KUKA KRL program: EPS_2_251349_MH90A_A_20250929014703.src

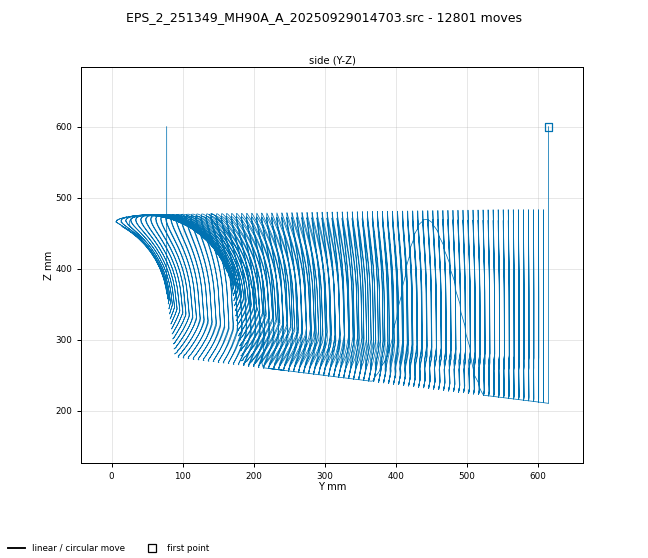
[picture p0: tool path of EPS_2_251349_MH90A_A_20250929014703.src, 12801 of 12803 moves have a stored position in this frame; points joined in program order, loops and branches not executed]
&ACCESS RVP
&REL 4
&COMMENT QRS 19112012
&PARAM EDITMASK = *
DEF PART()
EXT BAS (BAS_COMMAND :IN,REAL :IN )
INT I
BAS (#INITMOV,0 )

;KUKA QRS Post kuka4.cps  Date:22-06-2017 !

File_ID=2864

QRS_PRE_INIT()

;Init var - Until changes are made in qrs_pre_init
Outlet_Square_prg=0
Inlet_1_Square_prg=0
Inlet_2_Square_prg=0
Inlet_3_Square_prg=0
Inlet_4_Square_prg=0
Inlet_5_Square_prg=0

Outlet_1={X 0.000, Y 540.910, Z 382.500, B 0.000, E1 0.000 }
Inlet_1={X 0.000, Y 541.980, Z 367.500, B 0.000, E1 159.000 }
Outlet_1_type=201
Inlet_1_type=201
;QRS#1=Sidecore dimensions
;QRS#2=200-8" PVC SDR 35
;QRS#3=200-8" PVC SDR 35
;QRS#4=
;QRS#5=
;QRS#6=
;QRS#7=
;QRS#8=
;QRS#9=12-08 PSX
;QRS#10=12-08 PSX
;QRS#11=
;QRS#12=
;QRS#13=
;QRS#14=
;QRS#15=
;QRS#16=1220x127x762 2,5'
;QRS#17=EPS Height
;QRS#18=483
;QRS#19=*
;QRS#20= UPDATED VERSION 22-06-2017
;QRS#21=*
Outlet_Square=0100
Inlet_1_Square=0100
Inlet_2_Square=0
Inlet_3_Square=0
Inlet_4_Square=0
Inlet_5_Square=0
Mill_Square=1
Outlet_Square_Prg=204
Inlet_1_Square_prg=204

QRS_INIT()

$ADVANCE=5

; T1
PTP {E1 173.658,E2 173.658}
PTP {X 0,Y 615.42,A -85,B 0,C 180,E1 173.658,E2 173.658,E3 0,E4 0,E5 0,E6 0}
QRS_SPEED_INIT()
LIN {X 0,Y 615.42,Z 600,A -85,B 0,C 180,E1 173.658,E2 173.658,E3 0,E4 0,E5 0,E6 0} C_VEL
LIN {X 0,Y 615.42,Z 220.377,A -85,B 0,C 180,E1 173.658,E2 173.658} C_VEL
LIN {X 0,Y 615.42,Z 212.199,A -85,B 0,C 180,E1 173.658,E2 173.658} C_VEL
LIN {X 0,Y 615.409,Z 210.199,A -85,B 0,C 180,E1 173.472,E2 173.472} C_VEL
LIN {X 0,Y 615.414,Z 210.198,A -85,B 0,C 180,E1 171.465,E2 171.465} C_VEL
LIN {X 0,Y 615.421,Z 210.198,A -85,B 0,C 180,E1 169.475,E2 169.475} C_VEL
LIN {X 0,Y 615.428,Z 210.197,A -85,B 0,C 180,E1 167.472,E2 167.472} C_VEL
LIN {X 0,Y 615.434,Z 210.196,A -85,B 0,C 180,E1 165.453,E2 165.453} C_VEL
LIN {X 0,Y 615.439,Z 210.195,A -85,B 0,C 180,E1 163.415,E2 163.415} C_VEL
LIN {X 0,Y 615.442,Z 210.195,A -85,B 0,C 180,E1 161.356,E2 161.356} C_VEL
LIN {X 0,Y 615.442,Z 210.194,A -85,B 0,C 180,E1 159.271,E2 159.271} C_VEL
LIN {X 0,Y 615.441,Z 210.193,A -85,B 0,C 180,E1 157.157,E2 157.157} C_VEL
LIN {X 0,Y 615.437,Z 210.193,A -85,B 0,C 180,E1 155.01,E2 155.01} C_VEL
LIN {X 0,Y 615.432,Z 210.193,A -85,B 0,C 180,E1 152.824,E2 152.824} C_VEL
LIN {X 0,Y 615.429,Z 210.194,A -85,B 0,C 180,E1 150.595,E2 150.595} C_VEL
LIN {X 0,Y 615.43,Z 210.195,A -85,B 0,C 180,E1 148.316,E2 148.316} C_VEL
LIN {X 0,Y 615.446,Z 210.197,A -85,B 0,C 180,E1 145.98,E2 145.98} C_VEL
LIN {X 0,Y 615.487,Z 210.189,A -85,B 0,C 180,E1 143.061,E2 143.061} C_VEL
LIN {X 0,Y 615.489,Z 210.187,A -85,B 0,C 180,E1 140.935,E2 140.935} C_VEL
LIN {X 0,Y 615.457,Z 210.188,A -85,B 0,C 180,E1 138.529,E2 138.529} C_VEL
LIN {X 0,Y 615.441,Z 210.192,A -85,B 0,C 180,E1 136.005,E2 136.005} C_VEL
LIN {X 0,Y 615.49,Z 210.199,A -85,B 0,C 180,E1 133.243,E2 133.243} C_VEL
LIN {X 0,Y 615.493,Z 210.363,A -85,B 0,C 180,E1 131.038,E2 131.038} C_VEL
LIN {X 0,Y 615.491,Z 226.448,A -85,B 0,C 180,E1 128.483,E2 128.483} C_VEL
LIN {X 0,Y 615.431,Z 244.942,A -85,B 0,C 180,E1 125.618,E2 125.618} C_VEL
LIN {X 0,Y 615.451,Z 256.457,A -85,B 0,C 180,E1 123.87,E2 123.87} C_VEL
LIN {X 0,Y 615.447,Z 258.462,A -85,B 0,C 180,E1 123.794,E2 123.794} C_VEL
LIN {X 0,Y 615.497,Z 363.346,A -85,B 0,C 180,E1 122.552,E2 122.552} C_VEL
LIN {X 0,Y 615.5,Z 376.884,A -85,B 0,C 180,E1 122.258,E2 122.258} C_VEL
LIN {X 0,Y 615.498,Z 389.472,A -85,B 0,C 180,E1 121.847,E2 121.847} C_VEL
LIN {X 0,Y 615.478,Z 401.528,A -85,B 0,C 180,E1 121.313,E2 121.313} C_VEL
LIN {X 0,Y 615.477,Z 413.275,A -85,B 0,C 180,E1 120.633,E2 120.633} C_VEL
LIN {X 0,Y 615.497,Z 423.488,A -85,B 0,C 180,E1 119.894,E2 119.894} C_VEL
LIN {X 0,Y 615.497,Z 431.12,A -85,B 0,C 180,E1 119.217,E2 119.217} C_VEL
LIN {X 0,Y 615.497,Z 439.703,A -85,B 0,C 180,E1 118.324,E2 118.324} C_VEL
LIN {X 0,Y 615.488,Z 447.119,A -85,B 0,C 180,E1 117.36,E2 117.36} C_VEL
LIN {X 0,Y 615.496,Z 452.856,A -85,B 0,C 180,E1 116.442,E2 116.442} C_VEL
LIN {X 0,Y 615.495,Z 458.535,A -85,B 0,C 180,E1 115.285,E2 115.285} C_VEL
LIN {X 0,Y 615.496,Z 462.263,A -85,B 0,C 180,E1 114.27,E2 114.27} C_VEL
LIN {X 0,Y 615.494,Z 464.278,A -85,B 0,C 180,E1 113.555,E2 113.555} C_VEL
LIN {X 0,Y 615.492,Z 466.468,A -85,B 0,C 180,E1 112.359,E2 112.359} C_VEL
LIN {X 0,Y 615.497,Z 467.282,A -85,B 0,C 180,E1 111.43,E2 111.43} C_VEL
LIN {X 0,Y 615.494,Z 467.304,A -85,B 0,C 180,E1 110.572,E2 110.572} C_VEL
LIN {X 0,Y 615.496,Z 466.182,A -85,B 0,C 180,E1 109.336,E2 109.336} C_VEL
LIN {X 0,Y 615.496,Z 464.861,A -85,B 0,C 180,E1 108.622,E2 108.622} C_VEL
LIN {X 0,Y 615.499,Z 462.172,A -85,B 0,C 180,E1 107.612,E2 107.612} C_VEL
LIN {X 0,Y 615.495,Z 457.783,A -85,B 0,C 180,E1 106.45,E2 106.45} C_VEL
LIN {X 0,Y 615.497,Z 453.383,A -85,B 0,C 180,E1 105.564,E2 105.564} C_VEL
LIN {X 0,Y 615.489,Z 447.102,A -85,B 0,C 180,E1 104.548,E2 104.548} C_VEL
LIN {X 0,Y 615.5,Z 439.266,A -85,B 0,C 180,E1 103.536,E2 103.536} C_VEL
LIN {X 0,Y 615.496,Z 429.44,A -85,B 0,C 180,E1 102.529,E2 102.529} C_VEL
LIN {X 0,Y 615.498,Z 420.424,A -85,B 0,C 180,E1 101.776,E2 101.776} C_VEL
LIN {X 0,Y 615.475,Z 409.654,A -85,B 0,C 180,E1 101.049,E2 101.049} C_VEL
LIN {X 0,Y 615.492,Z 398.322,A -85,B 0,C 180,E1 100.443,E2 100.443} C_VEL
LIN {X 0,Y 615.498,Z 386.276,A -85,B 0,C 180,E1 99.944,E2 99.944} C_VEL
LIN {X 0,Y 615.498,Z 373.8,A -85,B 0,C 180,E1 99.57,E2 99.57} C_VEL
LIN {X 0,Y 615.497,Z 360.801,A -85,B 0,C 180,E1 99.322,E2 99.322} C_VEL
LIN {X 0,Y 615.431,Z 257.063,A -85,B 0,C 180,E1 98.082,E2 98.082} C_VEL
LIN {X 0,Y 615.443,Z 255.243,A -85,B 0,C 180,E1 97.875,E2 97.875} C_VEL
LIN {X 0,Y 615.472,Z 235.998,A -85,B 0,C 180,E1 94.912,E2 94.912} C_VEL
LIN {X 0,Y 615.489,Z 218.149,A -85,B 0,C 180,E1 92.126,E2 92.126} C_VEL
LIN {X 0,Y 615.493,Z 210.327,A -85,B 0,C 180,E1 90.858,E2 90.858} C_VEL
LIN {X 0,Y 615.425,Z 210.197,A -85,B 0,C 180,E1 88.036,E2 88.036} C_VEL
LIN {X 0,Y 615.43,Z 210.198,A -85,B 0,C 180,E1 86.07,E2 86.07} C_VEL
LIN {X 0,Y 615.436,Z 210.198,A -85,B 0,C 180,E1 84.1,E2 84.1} C_VEL
LIN {X 0,Y 615.444,Z 210.199,A -85,B 0,C 180,E1 82.123,E2 82.123} C_VEL
LIN {X 0,Y 615.449,Z 210.2,A -85,B 0,C 180,E1 80.136,E2 80.136} C_VEL
LIN {X 0,Y 615.413,Z 210.197,A -85,B 0,C 180,E1 77.467,E2 77.467} C_VEL
LIN {X 0,Y 615.414,Z 210.198,A -85,B 0,C 180,E1 75.448,E2 75.448} C_VEL
LIN {X 0,Y 615.411,Z 210.198,A -85,B 0,C 180,E1 73.41,E2 73.41} C_VEL
LIN {X 0,Y 615.412,Z 210.198,A -85,B 0,C 180,E1 71.351,E2 71.351} C_VEL
LIN {X 0,Y 615.411,Z 210.198,A -85,B 0,C 180,E1 69.266,E2 69.266} C_VEL
LIN {X 0,Y 615.409,Z 210.199,A -85,B 0,C 180,E1 67.152,E2 67.152} C_VEL
LIN {X 0,Y 615.407,Z 210.199,A -85,B 0,C 180,E1 65.004,E2 65.004} C_VEL
LIN {X 0,Y 615.404,Z 210.199,A -85,B 0,C 180,E1 62.818,E2 62.818} C_VEL
LIN {X 0,Y 615.442,Z 210.199,A -85,B 0,C 180,E1 60.204,E2 60.204} C_VEL
LIN {X 0,Y 615.467,Z 210.2,A -85,B 0,C 180,E1 57.54,E2 57.54} C_VEL
LIN {X 0,Y 615.43,Z 210.2,A -85,B 0,C 180,E1 55.18,E2 55.18} C_VEL
LIN {X 0,Y 615.405,Z 210.2,A -85,B 0,C 180,E1 52.751,E2 52.751} C_VEL
LIN {X 0,Y 615.408,Z 210.2,A -85,B 0,C 180,E1 50.243,E2 50.243} C_VEL
LIN {X 0,Y 615.426,Z 210.2,A -85,B 0,C 180,E1 47.92,E2 47.92} C_VEL
LIN {X 0,Y 615.448,Z 210.198,A -85,B 0,C 180,E1 44.927,E2 44.927} C_VEL
LIN {X 0,Y 615.473,Z 210.198,A -85,B 0,C 180,E1 43.045,E2 43.045} C_VEL
LIN {X 0,Y 615.432,Z 210.197,A -85,B 0,C 180,E1 40.606,E2 40.606} C_VEL
LIN {X 0,Y 615.48,Z 210.196,A -85,B 0,C 180,E1 38.9,E2 38.9} C_VEL
LIN {X 0,Y 615.432,Z 210.197,A -85,B 0,C 180,E1 36.424,E2 36.424} C_VEL
LIN {X 0,Y 615.414,Z 210.197,A -85,B 0,C 180,E1 34.022,E2 34.022} C_VEL
LIN {X 0,Y 615.415,Z 210.198,A -85,B 0,C 180,E1 31.685,E2 31.685} C_VEL
LIN {X 0,Y 615.423,Z 210.198,A -85,B 0,C 180,E1 29.405,E2 29.405} C_VEL
LIN {X 0,Y 615.453,Z 210.199,A -85,B 0,C 180,E1 27.037,E2 27.037} C_VEL
LIN {X 0,Y 615.44,Z 210.194,A -85,B 0,C 180,E1 23.997,E2 23.997} C_VEL
LIN {X 0,Y 615.464,Z 210.193,A -85,B 0,C 180,E1 22.134,E2 22.134} C_VEL
LIN {X 0,Y 615.462,Z 210.193,A -85,B 0,C 180,E1 20.03,E2 20.03} C_VEL
LIN {X 0,Y 615.459,Z 210.193,A -85,B 0,C 180,E1 17.954,E2 17.954} C_VEL
LIN {X 0,Y 615.467,Z 210.192,A -85,B 0,C 180,E1 15.902,E2 15.902} C_VEL
LIN {X 0,Y 615.425,Z 210.195,A -85,B 0,C 180,E1 13.199,E2 13.199} C_VEL
LIN {X 0,Y 615.426,Z 210.197,A -85,B 0,C 180,E1 10.856,E2 10.856} C_VEL
LIN {X 0,Y 615.446,Z 210.197,A -85,B 0,C 180,E1 8.534,E2 8.534} C_VEL
LIN {X 0,Y 615.497,Z 210.195,A -85,B 0,C 180,E1 5.896,E2 5.896} C_VEL
LIN {X 0,Y 615.453,Z 210.19,A -85,B 0,C 180,E1 3.27,E2 3.27} C_VEL
LIN {X 0,Y 615.466,Z 210.189,A -85,B 0,C 180,E1 1.306,E2 1.306} C_VEL
LIN {X 0,Y 615.432,Z 210.193,A -85,B 0,C 180,E1 -1.311,E2 -1.311} C_VEL
LIN {X 0,Y 615.436,Z 210.192,A -85,B 0,C 180,E1 -3.276,E2 -3.276} C_VEL
LIN {X 0,Y 615.441,Z 210.191,A -85,B 0,C 180,E1 -5.244,E2 -5.244} C_VEL
LIN {X 0,Y 615.449,Z 210.19,A -85,B 0,C 180,E1 -7.218,E2 -7.218} C_VEL
LIN {X 0,Y 615.457,Z 210.189,A -85,B 0,C 180,E1 -9.201,E2 -9.201} C_VEL
LIN {X 0,Y 615.466,Z 210.188,A -85,B 0,C 180,E1 -11.196,E2 -11.196} C_VEL
LIN {X 0,Y 615.472,Z 210.187,A -85,B 0,C 180,E1 -13.204,E2 -13.204} C_VEL
LIN {X 0,Y 615.439,Z 210.192,A -85,B 0,C 180,E1 -15.908,E2 -15.908} C_VEL
LIN {X 0,Y 615.475,Z 210.199,A -85,B 0,C 180,E1 -18.6,E2 -18.6} C_VEL
LIN {X 0,Y 615.485,Z 210.185,A -85,B 0,C 180,E1 -21.434,E2 -21.434} C_VEL
LIN {X 0,Y 615.446,Z 210.19,A -85,B 0,C 180,E1 -23.998,E2 -23.998} C_VEL
LIN {X 0,Y 615.447,Z 210.194,A -85,B 0,C 180,E1 -26.448,E2 -26.448} C_VEL
LIN {X 0,Y 615.493,Z 210.19,A -85,B 0,C 180,E1 -29.408,E2 -29.408} C_VEL
LIN {X 0,Y 615.489,Z 210.186,A -85,B 0,C 180,E1 -31.687,E2 -31.687} C_VEL
LIN {X 0,Y 615.474,Z 210.185,A -85,B 0,C 180,E1 -34.024,E2 -34.024} C_VEL
LIN {X 0,Y 615.453,Z 210.188,A -85,B 0,C 180,E1 -36.429,E2 -36.429} C_VEL
LIN {X 0,Y 615.461,Z 210.195,A -85,B 0,C 180,E1 -39.058,E2 -39.058} C_VEL
LIN {X 0,Y 615.491,Z 210.201,A -85,B 0,C 180,E1 -41.475,E2 -41.475} C_VEL
LIN {X 0,Y 615.496,Z 210.183,A -85,B 0,C 180,E1 -44.15,E2 -44.15} C_VEL
LIN {X 0,Y 615.454,Z 210.19,A -85,B 0,C 180,E1 -46.957,E2 -46.957} C_VEL
LIN {X 0,Y 615.464,Z 210.195,A -85,B 0,C 180,E1 -49.391,E2 -49.391} C_VEL
LIN {X 0,Y 615.49,Z 210.197,A -85,B 0,C 180,E1 -51.989,E2 -51.989} C_VEL
LIN {X 0,Y 615.489,Z 210.187,A -85,B 0,C 180,E1 -54.383,E2 -54.383} C_VEL
LIN {X 0,Y 615.486,Z 210.182,A -85,B 0,C 180,E1 -56.763,E2 -56.763} C_VEL
LIN {X 0,Y 615.472,Z 210.184,A -85,B 0,C 180,E1 -59.079,E2 -59.079} C_VEL
LIN {X 0,Y 615.46,Z 210.19,A -85,B 0,C 180,E1 -61.556,E2 -61.556} C_VEL
LIN {X 0,Y 615.498,Z 210.199,A -85,B 0,C 180,E1 -64.284,E2 -64.284} C_VEL
LIN {X 0,Y 615.484,Z 210.182,A -85,B 0,C 180,E1 -67.154,E2 -67.154} C_VEL
LIN {X 0,Y 615.492,Z 210.435,A -85,B 0,C 180,E1 -68.48,E2 -68.48} C_VEL
LIN {X 0,Y 615.494,Z 228.954,A -85,B 0,C 180,E1 -71.181,E2 -71.181} C_VEL
LIN {X 0,Y 615.488,Z 249.417,A -85,B 0,C 180,E1 -74.094,E2 -74.094} C_VEL
LIN {X 0,Y 615.473,Z 268.657,A -85,B 0,C 180,E1 -76.798,E2 -76.798} C_VEL
LIN {X 0,Y 615.487,Z 271.231,A -85,B 0,C 180,E1 -77.113,E2 -77.113} C_VEL
LIN {X 0,Y 615.49,Z 278.177,A -85,B 0,C 180,E1 -77.218,E2 -77.218} C_VEL
LIN {X 0,Y 615.498,Z 378.775,A -85,B 0,C 180,E1 -78.41,E2 -78.41} C_VEL
LIN {X 0,Y 615.498,Z 391.308,A -85,B 0,C 180,E1 -78.681,E2 -78.681} C_VEL
LIN {X 0,Y 615.496,Z 404.514,A -85,B 0,C 180,E1 -79.109,E2 -79.109} C_VEL
LIN {X 0,Y 615.491,Z 416.458,A -85,B 0,C 180,E1 -79.639,E2 -79.639} C_VEL
LIN {X 0,Y 615.48,Z 427.982,A -85,B 0,C 180,E1 -80.303,E2 -80.303} C_VEL
LIN {X 0,Y 615.499,Z 438.329,A -85,B 0,C 180,E1 -81.049,E2 -81.049} C_VEL
LIN {X 0,Y 615.498,Z 446.682,A -85,B 0,C 180,E1 -81.793,E2 -81.793} C_VEL
LIN {X 0,Y 615.498,Z 454.598,A -85,B 0,C 180,E1 -82.619,E2 -82.619} C_VEL
LIN {X 0,Y 615.49,Z 462.198,A -85,B 0,C 180,E1 -83.607,E2 -83.607} C_VEL
LIN {X 0,Y 615.498,Z 469.199,A -85,B 0,C 180,E1 -84.758,E2 -84.758} C_VEL
LIN {X 0,Y 615.493,Z 473.847,A -85,B 0,C 180,E1 -85.743,E2 -85.743} C_VEL
LIN {X 0,Y 615.494,Z 477.396,A -85,B 0,C 180,E1 -86.726,E2 -86.726} C_VEL
LIN {X 0,Y 615.497,Z 479.23,A -85,B 0,C 180,E1 -87.381,E2 -87.381} C_VEL
LIN {X 0,Y 615.497,Z 480.606,A -85,B 0,C 180,E1 -88.036,E2 -88.036} C_VEL
LIN {X 0,Y 615.496,Z 482.173,A -85,B 0,C 180,E1 -89.345,E2 -89.345} C_VEL
LIN {X 0,Y 615.494,Z 482.389,A -85,B 0,C 180,E1 -89.999,E2 -89.999} C_VEL
LIN {X 0,Y 615.495,Z 481.581,A -85,B 0,C 180,E1 -91.308,E2 -91.308} C_VEL
LIN {X 0,Y 615.497,Z 480.61,A -85,B 0,C 180,E1 -91.962,E2 -91.962} C_VEL
LIN {X 0,Y 615.497,Z 479.236,A -85,B 0,C 180,E1 -92.617,E2 -92.617} C_VEL
LIN {X 0,Y 615.496,Z 476.353,A -85,B 0,C 180,E1 -93.6,E2 -93.6} C_VEL
LIN {X 0,Y 615.498,Z 472.446,A -85,B 0,C 180,E1 -94.583,E2 -94.583} C_VEL
LIN {X 0,Y 615.499,Z 467.411,A -85,B 0,C 180,E1 -95.569,E2 -95.569} C_VEL
LIN {X 0,Y 615.489,Z 460.919,A -85,B 0,C 180,E1 -96.577,E2 -96.577} C_VEL
LIN {X 0,Y 615.497,Z 453.143,A -85,B 0,C 180,E1 -97.544,E2 -97.544} C_VEL
LIN {X 0,Y 615.498,Z 443.27,A -85,B 0,C 180,E1 -98.535,E2 -98.535} C_VEL
LIN {X 0,Y 615.495,Z 432.881,A -85,B 0,C 180,E1 -99.363,E2 -99.363} C_VEL
LIN {X 0,Y 615.475,Z 422.596,A -85,B 0,C 180,E1 -100.027,E2 -100.027} C_VEL
LIN {X 0,Y 615.497,Z 411.116,A -85,B 0,C 180,E1 -100.617,E2 -100.617} C_VEL
LIN {X 0,Y 615.499,Z 399.293,A -85,B 0,C 180,E1 -101.079,E2 -101.079} C_VEL
LIN {X 0,Y 615.498,Z 386.288,A -85,B 0,C 180,E1 -101.442,E2 -101.442} C_VEL
LIN {X 0,Y 615.5,Z 373.028,A -85,B 0,C 180,E1 -101.671,E2 -101.671} C_VEL
LIN {X 0,Y 615.488,Z 271.775,A -85,B 0,C 180,E1 -102.864,E2 -102.864} C_VEL
LIN {X 0,Y 615.485,Z 270.528,A -85,B 0,C 180,E1 -102.948,E2 -102.948} C_VEL
LIN {X 0,Y 615.481,Z 250.635,A -85,B 0,C 180,E1 -105.734,E2 -105.734} C_VEL
LIN {X 0,Y 615.491,Z 231.587,A -85,B 0,C 180,E1 -108.442,E2 -108.442} C_VEL
LIN {X 0,Y 615.493,Z 212.1,A -85,B 0,C 180,E1 -111.255,E2 -111.255} C_VEL
LIN {X 0,Y 615.49,Z 210.316,A -85,B 0,C 180,E1 -111.562,E2 -111.562} C_VEL
LIN {X 0,Y 615.461,Z 210.19,A -85,B 0,C 180,E1 -114.272,E2 -114.272} C_VEL
LIN {X 0,Y 615.497,Z 210.18,A -85,B 0,C 180,E1 -117.046,E2 -117.046} C_VEL
LIN {X 0,Y 615.497,Z 210.199,A -85,B 0,C 180,E1 -119.795,E2 -119.795} C_VEL
LIN {X 0,Y 615.457,Z 210.192,A -85,B 0,C 180,E1 -122.458,E2 -122.458} C_VEL
LIN {X 0,Y 615.455,Z 210.188,A -85,B 0,C 180,E1 -124.816,E2 -124.816} C_VEL
LIN {X 0,Y 615.476,Z 210.184,A -85,B 0,C 180,E1 -127.241,E2 -127.241} C_VEL
LIN {X 0,Y 615.498,Z 210.199,A -85,B 0,C 180,E1 -130.089,E2 -130.089} C_VEL
LIN {X 0,Y 615.48,Z 210.198,A -85,B 0,C 180,E1 -132.352,E2 -132.352} C_VEL
LIN {X 0,Y 615.443,Z 210.192,A -85,B 0,C 180,E1 -135.071,E2 -135.071} C_VEL
LIN {X 0,Y 615.498,Z 210.185,A -85,B 0,C 180,E1 -137.917,E2 -137.917} C_VEL
LIN {X 0,Y 615.495,Z 210.195,A -85,B 0,C 180,E1 -140.249,E2 -140.249} C_VEL
LIN {X 0,Y 615.443,Z 210.195,A -85,B 0,C 180,E1 -143.066,E2 -143.066} C_VEL
LIN {X 0,Y 615.437,Z 210.193,A -85,B 0,C 180,E1 -145.304,E2 -145.304} C_VEL
LIN {X 0,Y 615.44,Z 210.191,A -85,B 0,C 180,E1 -147.673,E2 -147.673} C_VEL
LIN {X 0,Y 615.491,Z 210.198,A -85,B 0,C 180,E1 -150.592,E2 -150.592} C_VEL
LIN {X 0,Y 615.473,Z 210.199,A -85,B 0,C 180,E1 -152.954,E2 -152.954} C_VEL
LIN {X 0,Y 615.473,Z 210.199,A -85,B 0,C 180,E1 -155.006,E2 -155.006} C_VEL
LIN {X 0,Y 615.427,Z 210.196,A -85,B 0,C 180,E1 -157.664,E2 -157.664} C_VEL
LIN {X 0,Y 615.423,Z 210.195,A -85,B 0,C 180,E1 -159.963,E2 -159.963} C_VEL
LIN {X 0,Y 615.48,Z 210.193,A -85,B 0,C 180,E1 -162.727,E2 -162.727} C_VEL
LIN {X 0,Y 615.452,Z 210.199,A -85,B 0,C 180,E1 -165.448,E2 -165.448} C_VEL
LIN {X 0,Y 615.455,Z 210.199,A -85,B 0,C 180,E1 -167.467,E2 -167.467} C_VEL
LIN {X 0,Y 615.462,Z 210.199,A -85,B 0,C 180,E1 -169.47,E2 -169.47} C_VEL
LIN {X 0,Y 615.413,Z 210.198,A -85,B 0,C 180,E1 -172.121,E2 -172.121} C_VEL
LIN {X 0,Y 615.413,Z 210.199,A -85,B 0,C 180,E1 -174.098,E2 -174.098} C_VEL
LIN {X 0,Y 615.417,Z 210.199,A -85,B 0,C 180,E1 -176.069,E2 -176.069} C_VEL
LIN {X 0,Y 615.419,Z 210.2,A -85,B 0,C 180,E1 -178.034,E2 -178.034} C_VEL
LIN {X 0,Y 615.43,Z 210.2,A -85,B 0,C 180,E1 -179.997,E2 -179.997} C_VEL
LIN {X 0,Y 615.44,Z 210.2,A -85,B 0,C 180,E1 -181.961,E2 -181.961} C_VEL
LIN {X 0,Y 615.404,Z 210.2,A -85,B 0,C 180,E1 -184.582,E2 -184.582} C_VEL
LIN {X 0,Y 615.409,Z 210.199,A -85,B 0,C 180,E1 -186.528,E2 -186.528} C_VEL
LIN {X 0,Y 614.74,Z 210.347,A -85,B 0,C 180,E1 -187.074,E2 -187.074} C_VEL
LIN {X 0,Y 611.905,Z 210.764,A -85,B 0,C 180,E1 -187.961,E2 -187.961} C_VEL
LIN {X 0,Y 609.519,Z 211.07,A -85,B 0,C 180,E1 -188.673,E2 -188.673} C_VEL
LIN {X 0,Y 608.5,Z 211.185,A -85,B 0,C 180,E1 -189.223,E2 -189.223} C_VEL
LIN {X 0,Y 608.42,Z 211.194,A -85,B 0,C 180,E1 -189.409,E2 -189.409} C_VEL
LIN {X 0,Y 608.446,Z 211.196,A -85,B 0,C 180,E1 -191.997,E2 -191.997} C_VEL
LIN {X 0,Y 608.393,Z 211.194,A -85,B 0,C 180,E1 -194.719,E2 -194.719} C_VEL
LIN {X 0,Y 608.401,Z 211.193,A -85,B 0,C 180,E1 -196.782,E2 -196.782} C_VEL
LIN {X 0,Y 608.415,Z 211.191,A -85,B 0,C 180,E1 -198.867,E2 -198.867} C_VEL
LIN {X 0,Y 608.411,Z 211.192,A -85,B 0,C 180,E1 -200.98,E2 -200.98} C_VEL
LIN {X 0,Y 608.403,Z 211.193,A -85,B 0,C 180,E1 -203.122,E2 -203.122} C_VEL
LIN {X 0,Y 608.396,Z 211.193,A -85,B 0,C 180,E1 -205.3,E2 -205.3} C_VEL
LIN {X 0,Y 608.407,Z 211.193,A -85,B 0,C 180,E1 -207.516,E2 -207.516} C_VEL
LIN {X 0,Y 608.428,Z 211.194,A -85,B 0,C 180,E1 -209.968,E2 -209.968} C_VEL
LIN {X 0,Y 608.437,Z 211.192,A -85,B 0,C 180,E1 -212.876,E2 -212.876} C_VEL
LIN {X 0,Y 608.417,Z 211.191,A -85,B 0,C 180,E1 -215.275,E2 -215.275} C_VEL
LIN {X 0,Y 608.431,Z 211.189,A -85,B 0,C 180,E1 -217.744,E2 -217.744} C_VEL
LIN {X 0,Y 608.444,Z 211.193,A -85,B 0,C 180,E1 -220.33,E2 -220.33} C_VEL
LIN {X 0,Y 608.472,Z 211.186,A -85,B 0,C 180,E1 -223.311,E2 -223.311} C_VEL
LIN {X 0,Y 608.433,Z 211.19,A -85,B 0,C 180,E1 -226.129,E2 -226.129} C_VEL
LIN {X 0,Y 608.493,Z 211.363,A -85,B 0,C 180,E1 -228.883,E2 -228.883} C_VEL
LIN {X 0,Y 608.497,Z 226.062,A -85,B 0,C 180,E1 -231.237,E2 -231.237} C_VEL
LIN {X 0,Y 608.436,Z 244.625,A -85,B 0,C 180,E1 -234.142,E2 -234.142} C_VEL
LIN {X 0,Y 608.459,Z 256.853,A -85,B 0,C 180,E1 -236.006,E2 -236.006} C_VEL
LIN {X 0,Y 608.526,Z 259.752,A -85,B 0,C 180,E1 -236.073,E2 -236.073} C_VEL
LIN {X 0,Y 608.562,Z 364.518,A -85,B 0,C 180,E1 -237.332,E2 -237.332} C_VEL
LIN {X 0,Y 608.549,Z 378.086,A -85,B 0,C 180,E1 -237.641,E2 -237.641} C_VEL
LIN {X 0,Y 608.528,Z 390.418,A -85,B 0,C 180,E1 -238.057,E2 -238.057} C_VEL
LIN {X 0,Y 608.481,Z 402.109,A -85,B 0,C 180,E1 -238.589,E2 -238.589} C_VEL
LIN {X 0,Y 608.49,Z 413.644,A -85,B 0,C 180,E1 -239.266,E2 -239.266} C_VEL
LIN {X 0,Y 608.485,Z 424.769,A -85,B 0,C 180,E1 -240.085,E2 -240.085} C_VEL
LIN {X 0,Y 608.485,Z 434.427,A -85,B 0,C 180,E1 -240.982,E2 -240.982} C_VEL
LIN {X 0,Y 608.45,Z 442.773,A -85,B 0,C 180,E1 -241.922,E2 -241.922} C_VEL
LIN {X 0,Y 608.435,Z 449.046,A -85,B 0,C 180,E1 -242.791,E2 -242.791} C_VEL
LIN {X 0,Y 608.45,Z 453.885,A -85,B 0,C 180,E1 -243.597,E2 -243.597} C_VEL
LIN {X 0,Y 608.442,Z 459.203,A -85,B 0,C 180,E1 -244.7,E2 -244.7} C_VEL
LIN {X 0,Y 608.425,Z 463.318,A -85,B 0,C 180,E1 -245.847,E2 -245.847} C_VEL
LIN {X 0,Y 608.427,Z 465.861,A -85,B 0,C 180,E1 -246.876,E2 -246.876} C_VEL
LIN {X 0,Y 608.428,Z 467.034,A -85,B 0,C 180,E1 -247.594,E2 -247.594} C_VEL
LIN {X 0,Y 608.416,Z 467.73,A -85,B 0,C 180,E1 -248.308,E2 -248.308} C_VEL
LIN {X 0,Y 608.429,Z 467.942,A -85,B 0,C 180,E1 -249.318,E2 -249.318} C_VEL
LIN {X 0,Y 608.417,Z 467.112,A -85,B 0,C 180,E1 -250.43,E2 -250.43} C_VEL
LIN {X 0,Y 608.439,Z 465.721,A -85,B 0,C 180,E1 -251.278,E2 -251.278} C_VEL
LIN {X 0,Y 608.427,Z 462.42,A -85,B 0,C 180,E1 -252.524,E2 -252.524} C_VEL
LIN {X 0,Y 608.428,Z 458.874,A -85,B 0,C 180,E1 -253.467,E2 -253.467} C_VEL
LIN {X 0,Y 608.458,Z 453.327,A -85,B 0,C 180,E1 -254.595,E2 -254.595} C_VEL
LIN {X 0,Y 608.455,Z 446.87,A -85,B 0,C 180,E1 -255.622,E2 -255.622} C_VEL
LIN {X 0,Y 608.479,Z 438.77,A -85,B 0,C 180,E1 -256.645,E2 -256.645} C_VEL
LIN {X 0,Y 608.466,Z 428.738,A -85,B 0,C 180,E1 -257.663,E2 -257.663} C_VEL
LIN {X 0,Y 608.502,Z 418.214,A -85,B 0,C 180,E1 -258.509,E2 -258.509} C_VEL
LIN {X 0,Y 608.482,Z 407.89,A -85,B 0,C 180,E1 -259.182,E2 -259.182} C_VEL
LIN {X 0,Y 608.53,Z 396.519,A -85,B 0,C 180,E1 -259.773,E2 -259.773} C_VEL
LIN {X 0,Y 608.549,Z 384.936,A -85,B 0,C 180,E1 -260.235,E2 -260.235} C_VEL
LIN {X 0,Y 608.559,Z 371.678,A -85,B 0,C 180,E1 -260.613,E2 -260.613} C_VEL
LIN {X 0,Y 608.566,Z 358.741,A -85,B 0,C 180,E1 -260.843,E2 -260.843} C_VEL
LIN {X 0,Y 608.486,Z 257.37,A -85,B 0,C 180,E1 -262.055,E2 -262.055} C_VEL
LIN {X 0,Y 608.415,Z 255.913,A -85,B 0,C 180,E1 -262.2,E2 -262.2} C_VEL
LIN {X 0,Y 608.492,Z 237.665,A -85,B 0,C 180,E1 -265.032,E2 -265.032} C_VEL
LIN {X 0,Y 608.498,Z 219.765,A -85,B 0,C 180,E1 -267.85,E2 -267.85} C_VEL
LIN {X 0,Y 608.465,Z 211.285,A -85,B 0,C 180,E1 -269.236,E2 -269.236} C_VEL
LIN {X 0,Y 608.396,Z 211.195,A -85,B 0,C 180,E1 -271.987,E2 -271.987} C_VEL
LIN {X 0,Y 608.398,Z 211.195,A -85,B 0,C 180,E1 -273.975,E2 -273.975} C_VEL
LIN {X 0,Y 608.408,Z 211.194,A -85,B 0,C 180,E1 -275.968,E2 -275.968} C_VEL
LIN {X 0,Y 608.432,Z 211.192,A -85,B 0,C 180,E1 -277.969,E2 -277.969} C_VEL
LIN {X 0,Y 608.413,Z 211.195,A -85,B 0,C 180,E1 -279.979,E2 -279.979} C_VEL
LIN {X 0,Y 608.424,Z 211.194,A -85,B 0,C 180,E1 -282.001,E2 -282.001} C_VEL
LIN {X 0,Y 608.385,Z 211.195,A -85,B 0,C 180,E1 -284.724,E2 -284.724} C_VEL
LIN {X 0,Y 608.417,Z 211.196,A -85,B 0,C 180,E1 -287.479,E2 -287.479} C_VEL
LIN {X 0,Y 608.421,Z 211.195,A -85,B 0,C 180,E1 -290.276,E2 -290.276} C_VEL
LIN {X 0,Y 608.418,Z 211.193,A -85,B 0,C 180,E1 -292.479,E2 -292.479} C_VEL
LIN {X 0,Y 608.404,Z 211.195,A -85,B 0,C 180,E1 -294.574,E2 -294.574} C_VEL
LIN {X 0,Y 608.384,Z 211.195,A -85,B 0,C 180,E1 -297.2,E2 -297.2} C_VEL
LIN {X 0,Y 608.462,Z 211.192,A -85,B 0,C 180,E1 -299.98,E2 -299.98} C_VEL
LIN {X 0,Y 608.405,Z 211.194,A -85,B 0,C 180,E1 -302.884,E2 -302.884} C_VEL
LIN {X 0,Y 608.378,Z 211.196,A -85,B 0,C 180,E1 -305.283,E2 -305.283} C_VEL
LIN {X 0,Y 608.422,Z 211.197,A -85,B 0,C 180,E1 -308.242,E2 -308.242} C_VEL
LIN {X 0,Y 608.391,Z 211.196,A -85,B 0,C 180,E1 -311.183,E2 -311.183} C_VEL
LIN {X 0,Y 608.405,Z 211.193,A -85,B 0,C 180,E1 -313.876,E2 -313.876} C_VEL
LIN {X 0,Y 608.478,Z 211.194,A -85,B 0,C 180,E1 -316.691,E2 -316.691} C_VEL
LIN {X 0,Y 608.41,Z 211.192,A -85,B 0,C 180,E1 -319.677,E2 -319.677} C_VEL
LIN {X 0,Y 608.413,Z 211.192,A -85,B 0,C 180,E1 -322.255,E2 -322.255} C_VEL
LIN {X 0,Y 608.447,Z 211.197,A -85,B 0,C 180,E1 -325.096,E2 -325.096} C_VEL
LIN {X 0,Y 608.415,Z 211.191,A -85,B 0,C 180,E1 -327.907,E2 -327.907} C_VEL
LIN {X 0,Y 608.402,Z 211.193,A -85,B 0,C 180,E1 -330.221,E2 -330.221} C_VEL
LIN {X 0,Y 608.402,Z 211.193,A -85,B 0,C 180,E1 -332.484,E2 -332.484} C_VEL
LIN {X 0,Y 608.432,Z 211.199,A -85,B 0,C 180,E1 -335.432,E2 -335.432} C_VEL
LIN {X 0,Y 608.423,Z 211.19,A -85,B 0,C 180,E1 -338.31,E2 -338.31} C_VEL
LIN {X 0,Y 608.406,Z 211.192,A -85,B 0,C 180,E1 -340.431,E2 -340.431} C_VEL
LIN {X 0,Y 608.419,Z 211.195,A -85,B 0,C 180,E1 -343.218,E2 -343.218} C_VEL
LIN {X 0,Y 608.472,Z 211.19,A -85,B 0,C 180,E1 -345.984,E2 -345.984} C_VEL
LIN {X 0,Y 608.412,Z 211.191,A -85,B 0,C 180,E1 -348.678,E2 -348.678} C_VEL
LIN {X 0,Y 608.428,Z 211.189,A -85,B 0,C 180,E1 -350.697,E2 -350.697} C_VEL
LIN {X 0,Y 608.418,Z 211.191,A -85,B 0,C 180,E1 -352.703,E2 -352.703} C_VEL
LIN {X 0,Y 608.43,Z 211.19,A -85,B 0,C 180,E1 -354.701,E2 -354.701} C_VEL
LIN {X 0,Y 608.429,Z 211.19,A -85,B 0,C 180,E1 -357.354,E2 -357.354} C_VEL
LIN {X 0,Y 608.469,Z 211.193,A -85,B 0,C 180,E1 -360.003,E2 -360.003} C_VEL
LIN {X 0,Y 608.48,Z 211.187,A -85,B 0,C 180,E1 -362.65,E2 -362.65} C_VEL
LIN {X 0,Y 608.424,Z 211.19,A -85,B 0,C 180,E1 -365.305,E2 -365.305} C_VEL
LIN {X 0,Y 608.423,Z 211.19,A -85,B 0,C 180,E1 -367.302,E2 -367.302} C_VEL
LIN {X 0,Y 608.441,Z 211.188,A -85,B 0,C 180,E1 -369.308,E2 -369.308} C_VEL
LIN {X 0,Y 608.432,Z 211.189,A -85,B 0,C 180,E1 -371.327,E2 -371.327} C_VEL
LIN {X 0,Y 608.444,Z 211.188,A -85,B 0,C 180,E1 -373.359,E2 -373.359} C_VEL
LIN {X 0,Y 608.456,Z 211.186,A -85,B 0,C 180,E1 -375.408,E2 -375.408} C_VEL
LIN {X 0,Y 608.416,Z 211.193,A -85,B 0,C 180,E1 -378.175,E2 -378.175} C_VEL
LIN {X 0,Y 608.459,Z 211.194,A -85,B 0,C 180,E1 -380.983,E2 -380.983} C_VEL
LIN {X 0,Y 608.44,Z 211.188,A -85,B 0,C 180,E1 -383.848,E2 -383.848} C_VEL
LIN {X 0,Y 608.425,Z 211.19,A -85,B 0,C 180,E1 -386.038,E2 -386.038} C_VEL
LIN {X 0,Y 608.416,Z 211.191,A -85,B 0,C 180,E1 -388.27,E2 -388.27} C_VEL
LIN {X 0,Y 608.43,Z 211.191,A -85,B 0,C 180,E1 -390.549,E2 -390.549} C_VEL
LIN {X 0,Y 608.445,Z 211.192,A -85,B 0,C 180,E1 -392.882,E2 -392.882} C_VEL
LIN {X 0,Y 608.437,Z 211.2,A -85,B 0,C 180,E1 -395.28,E2 -395.28} C_VEL
LIN {X 0,Y 608.467,Z 211.189,A -85,B 0,C 180,E1 -397.748,E2 -397.748} C_VEL
LIN {X 0,Y 608.445,Z 211.187,A -85,B 0,C 180,E1 -400.327,E2 -400.327} C_VEL
LIN {X 0,Y 608.423,Z 211.192,A -85,B 0,C 180,E1 -402.964,E2 -402.964} C_VEL
LIN {X 0,Y 608.458,Z 211.196,A -85,B 0,C 180,E1 -405.737,E2 -405.737} C_VEL
LIN {X 0,Y 608.449,Z 211.187,A -85,B 0,C 180,E1 -408.661,E2 -408.661} C_VEL
LIN {X 0,Y 608.426,Z 211.194,A -85,B 0,C 180,E1 -411.408,E2 -411.408} C_VEL
LIN {X 0,Y 608.453,Z 211.197,A -85,B 0,C 180,E1 -413.955,E2 -413.955} C_VEL
LIN {X 0,Y 608.457,Z 211.191,A -85,B 0,C 180,E1 -416.328,E2 -416.328} C_VEL
LIN {X 0,Y 608.454,Z 211.187,A -85,B 0,C 180,E1 -418.733,E2 -418.733} C_VEL
LIN {X 0,Y 608.454,Z 211.187,A -85,B 0,C 180,E1 -421.385,E2 -421.385} C_VEL
LIN {X 0,Y 608.44,Z 211.194,A -85,B 0,C 180,E1 -423.963,E2 -423.963} C_VEL
LIN {X 0,Y 608.451,Z 211.19,A -85,B 0,C 180,E1 -426.875,E2 -426.875} C_VEL
LIN {X 0,Y 608.471,Z 211.348,A -85,B 0,C 180,E1 -428.352,E2 -428.352} C_VEL
LIN {X 0,Y 608.512,Z 222.951,A -85,B 0,C 180,E1 -430.079,E2 -430.079} C_VEL
LIN {X 0,Y 608.519,Z 242.257,A -85,B 0,C 180,E1 -432.871,E2 -432.871} C_VEL
LIN {X 0,Y 608.482,Z 262.77,A -85,B 0,C 180,E1 -435.791,E2 -435.791} C_VEL
LIN {X 0,Y 608.497,Z 271.278,A -85,B 0,C 180,E1 -436.962,E2 -436.962} C_VEL
LIN {X 0,Y 608.588,Z 276.429,A -85,B 0,C 180,E1 -437.049,E2 -437.049} C_VEL
LIN {X 0,Y 608.549,Z 378.895,A -85,B 0,C 180,E1 -438.276,E2 -438.276} C_VEL
LIN {X 0,Y 608.548,Z 392.182,A -85,B 0,C 180,E1 -438.571,E2 -438.571} C_VEL
LIN {X 0,Y 608.545,Z 405.333,A -85,B 0,C 180,E1 -439.009,E2 -439.009} C_VEL
LIN {X 0,Y 608.516,Z 416.616,A -85,B 0,C 180,E1 -439.518,E2 -439.518} C_VEL
LIN {X 0,Y 608.468,Z 428.183,A -85,B 0,C 180,E1 -440.19,E2 -440.19} C_VEL
LIN {X 0,Y 608.485,Z 438.582,A -85,B 0,C 180,E1 -440.945,E2 -440.945} C_VEL
LIN {X 0,Y 608.459,Z 446.993,A -85,B 0,C 180,E1 -441.698,E2 -441.698} C_VEL
LIN {X 0,Y 608.471,Z 454.952,A -85,B 0,C 180,E1 -442.533,E2 -442.533} C_VEL
LIN {X 0,Y 608.437,Z 462.299,A -85,B 0,C 180,E1 -443.486,E2 -443.486} C_VEL
LIN {X 0,Y 608.45,Z 467.86,A -85,B 0,C 180,E1 -444.365,E2 -444.365} C_VEL
LIN {X 0,Y 608.432,Z 472.946,A -85,B 0,C 180,E1 -445.361,E2 -445.361} C_VEL
LIN {X 0,Y 608.449,Z 476.893,A -85,B 0,C 180,E1 -446.357,E2 -446.357} C_VEL
LIN {X 0,Y 608.425,Z 479.807,A -85,B 0,C 180,E1 -447.351,E2 -447.351} C_VEL
LIN {X 0,Y 608.442,Z 481.2,A -85,B 0,C 180,E1 -448.013,E2 -448.013} C_VEL
LIN {X 0,Y 608.439,Z 482.783,A -85,B 0,C 180,E1 -449.337,E2 -449.337} C_VEL
LIN {X 0,Y 608.434,Z 483,A -85,B 0,C 180,E1 -449.999,E2 -449.999} C_VEL
LIN {X 0,Y 608.448,Z 482.185,A -85,B 0,C 180,E1 -451.323,E2 -451.323} C_VEL
LIN {X 0,Y 608.442,Z 481.203,A -85,B 0,C 180,E1 -451.985,E2 -451.985} C_VEL
LIN {X 0,Y 608.425,Z 479.812,A -85,B 0,C 180,E1 -452.647,E2 -452.647} C_VEL
LIN {X 0,Y 608.449,Z 476.9,A -85,B 0,C 180,E1 -453.641,E2 -453.641} C_VEL
LIN {X 0,Y 608.432,Z 472.955,A -85,B 0,C 180,E1 -454.637,E2 -454.637} C_VEL
LIN {X 0,Y 608.437,Z 466.883,A -85,B 0,C 180,E1 -455.8,E2 -455.8} C_VEL
LIN {X 0,Y 608.461,Z 460.243,A -85,B 0,C 180,E1 -456.798,E2 -456.798} C_VEL
LIN {X 0,Y 608.455,Z 451.999,A -85,B 0,C 180,E1 -457.799,E2 -457.799} C_VEL
LIN {X 0,Y 608.477,Z 441.611,A -85,B 0,C 180,E1 -458.802,E2 -458.802} C_VEL
LIN {X 0,Y 608.486,Z 430.764,A -85,B 0,C 180,E1 -459.64,E2 -459.64} C_VEL
LIN {X 0,Y 608.489,Z 419.795,A -85,B 0,C 180,E1 -460.312,E2 -460.312} C_VEL
LIN {X 0,Y 608.536,Z 407.802,A -85,B 0,C 180,E1 -460.889,E2 -460.889} C_VEL
LIN {X 0,Y 608.533,Z 395.914,A -85,B 0,C 180,E1 -461.322,E2 -461.322} C_VEL
LIN {X 0,Y 608.542,Z 383.573,A -85,B 0,C 180,E1 -461.638,E2 -461.638} C_VEL
LIN {X 0,Y 608.574,Z 367.83,A -85,B 0,C 180,E1 -461.87,E2 -461.87} C_VEL
LIN {X 0,Y 608.547,Z 271.79,A -85,B 0,C 180,E1 -463.014,E2 -463.014} C_VEL
LIN {X 0,Y 608.459,Z 270.66,A -85,B 0,C 180,E1 -463.1,E2 -463.1} C_VEL
LIN {X 0,Y 608.491,Z 251.925,A -85,B 0,C 180,E1 -465.748,E2 -465.748} C_VEL
LIN {X 0,Y 608.512,Z 232.759,A -85,B 0,C 180,E1 -468.497,E2 -468.497} C_VEL
LIN {X 0,Y 608.571,Z 213.314,A -85,B 0,C 180,E1 -471.331,E2 -471.331} C_VEL
LIN {X 0,Y 608.478,Z 211.266,A -85,B 0,C 180,E1 -471.69,E2 -471.69} C_VEL
LIN {X 0,Y 608.444,Z 211.188,A -85,B 0,C 180,E1 -474.57,E2 -474.57} C_VEL
LIN {X 0,Y 608.486,Z 211.185,A -85,B 0,C 180,E1 -477.207,E2 -477.207} C_VEL
LIN {X 0,Y 608.452,Z 211.196,A -85,B 0,C 180,E1 -479.968,E2 -479.968} C_VEL
LIN {X 0,Y 608.437,Z 211.19,A -85,B 0,C 180,E1 -482.518,E2 -482.518} C_VEL
LIN {X 0,Y 608.425,Z 211.19,A -85,B 0,C 180,E1 -484.901,E2 -484.901} C_VEL
LIN {X 0,Y 608.467,Z 211.19,A -85,B 0,C 180,E1 -487.745,E2 -487.745} C_VEL
LIN {X 0,Y 608.442,Z 211.196,A -85,B 0,C 180,E1 -490.327,E2 -490.327} C_VEL
LIN {X 0,Y 608.419,Z 211.191,A -85,B 0,C 180,E1 -492.961,E2 -492.961} C_VEL
LIN {X 0,Y 608.459,Z 211.188,A -85,B 0,C 180,E1 -495.734,E2 -495.734} C_VEL
LIN {X 0,Y 608.441,Z 211.194,A -85,B 0,C 180,E1 -498.658,E2 -498.658} C_VEL
LIN {X 0,Y 608.41,Z 211.192,A -85,B 0,C 180,E1 -501.406,E2 -501.406} C_VEL
LIN {X 0,Y 608.443,Z 211.19,A -85,B 0,C 180,E1 -503.952,E2 -503.952} C_VEL
LIN {X 0,Y 608.465,Z 211.191,A -85,B 0,C 180,E1 -506.328,E2 -506.328} C_VEL
LIN {X 0,Y 608.439,Z 211.198,A -85,B 0,C 180,E1 -508.731,E2 -508.731} C_VEL
LIN {X 0,Y 608.428,Z 211.191,A -85,B 0,C 180,E1 -511.385,E2 -511.385} C_VEL
LIN {X 0,Y 608.416,Z 211.195,A -85,B 0,C 180,E1 -513.222,E2 -513.222} C_VEL
LIN {X 0,Y 608.419,Z 211.193,A -85,B 0,C 180,E1 -515.426,E2 -515.426} C_VEL
LIN {X 0,Y 608.445,Z 211.189,A -85,B 0,C 180,E1 -518.306,E2 -518.306} C_VEL
LIN {X 0,Y 608.445,Z 211.193,A -85,B 0,C 180,E1 -521.287,E2 -521.287} C_VEL
LIN {X 0,Y 608.404,Z 211.193,A -85,B 0,C 180,E1 -523.903,E2 -523.903} C_VEL
LIN {X 0,Y 608.434,Z 211.191,A -85,B 0,C 180,E1 -526.641,E2 -526.641} C_VEL
LIN {X 0,Y 608.449,Z 211.196,A -85,B 0,C 180,E1 -529.348,E2 -529.348} C_VEL
LIN {X 0,Y 608.388,Z 211.195,A -85,B 0,C 180,E1 -532.03,E2 -532.03} C_VEL
LIN {X 0,Y 608.396,Z 211.195,A -85,B 0,C 180,E1 -534.03,E2 -534.03} C_VEL
LIN {X 0,Y 608.391,Z 211.196,A -85,B 0,C 180,E1 -536.023,E2 -536.023} C_VEL
LIN {X 0,Y 608.394,Z 211.196,A -85,B 0,C 180,E1 -538.012,E2 -538.012} C_VEL
LIN {X 0,Y 608.424,Z 211.193,A -85,B 0,C 180,E1 -539.997,E2 -539.997} C_VEL
LIN {X 0,Y 608.4,Z 211.193,A -85,B 0,C 180,E1 -542.646,E2 -542.646} C_VEL
LIN {X 0,Y 608.419,Z 211.195,A -85,B 0,C 180,E1 -545.299,E2 -545.299} C_VEL
LIN {X 0,Y 608.459,Z 211.193,A -85,B 0,C 180,E1 -547.964,E2 -547.964} C_VEL
LIN {X 0,Y 608.42,Z 211.194,A -85,B 0,C 180,E1 -549.409,E2 -549.409} C_VEL
LIN {X 0,Y 607.768,Z 211.281,A -85,B 0,C 180,E1 -549.962,E2 -549.962} C_VEL
LIN {X 0,Y 604.935,Z 211.634,A -85,B 0,C 180,E1 -550.859,E2 -550.859} C_VEL
LIN {X 0,Y 602.522,Z 211.935,A -85,B 0,C 180,E1 -551.58,E2 -551.58} C_VEL
LIN {X 0,Y 601.465,Z 212.064,A -85,B 0,C 180,E1 -552.136,E2 -552.136} C_VEL
LIN {X 0,Y 601.369,Z 212.072,A -85,B 0,C 180,E1 -552.325,E2 -552.325} C_VEL
LIN {X 0,Y 601.363,Z 212.07,A -85,B 0,C 180,E1 -554.895,E2 -554.895} C_VEL
LIN {X 0,Y 601.376,Z 212.068,A -85,B 0,C 180,E1 -556.984,E2 -556.984} C_VEL
LIN {X 0,Y 601.376,Z 212.074,A -85,B 0,C 180,E1 -559.807,E2 -559.807} C_VEL
LIN {X 0,Y 601.395,Z 212.068,A -85,B 0,C 180,E1 -562.68,E2 -562.68} C_VEL
LIN {X 0,Y 601.368,Z 212.07,A -85,B 0,C 180,E1 -564.876,E2 -564.876} C_VEL
LIN {X 0,Y 601.361,Z 212.07,A -85,B 0,C 180,E1 -567.356,E2 -567.356} C_VEL
LIN {X 0,Y 601.381,Z 212.067,A -85,B 0,C 180,E1 -569.391,E2 -569.391} C_VEL
LIN {X 0,Y 601.373,Z 212.07,A -85,B 0,C 180,E1 -571.724,E2 -571.724} C_VEL
LIN {X 0,Y 601.396,Z 212.07,A -85,B 0,C 180,E1 -574.116,E2 -574.116} C_VEL
LIN {X 0,Y 601.397,Z 212.077,A -85,B 0,C 180,E1 -576.578,E2 -576.578} C_VEL
LIN {X 0,Y 601.408,Z 212.064,A -85,B 0,C 180,E1 -579.534,E2 -579.534} C_VEL
LIN {X 0,Y 601.39,Z 212.067,A -85,B 0,C 180,E1 -581.763,E2 -581.763} C_VEL
LIN {X 0,Y 601.384,Z 212.074,A -85,B 0,C 180,E1 -584.533,E2 -584.533} C_VEL
LIN {X 0,Y 601.408,Z 212.069,A -85,B 0,C 180,E1 -587.403,E2 -587.403} C_VEL
LIN {X 0,Y 601.456,Z 212.321,A -85,B 0,C 180,E1 -588.798,E2 -588.798} C_VEL
LIN {X 0,Y 601.489,Z 225.181,A -85,B 0,C 180,E1 -590.881,E2 -590.881} C_VEL
LIN {X 0,Y 601.441,Z 243.117,A -85,B 0,C 180,E1 -593.727,E2 -593.727} C_VEL
LIN {X 0,Y 601.444,Z 256.957,A -85,B 0,C 180,E1 -595.859,E2 -595.859} C_VEL
LIN {X 0,Y 601.619,Z 261.132,A -85,B 0,C 180,E1 -595.938,E2 -595.938} C_VEL
LIN {X 0,Y 601.628,Z 364.45,A -85,B 0,C 180,E1 -597.194,E2 -597.194} C_VEL
LIN {X 0,Y 601.605,Z 377.676,A -85,B 0,C 180,E1 -597.496,E2 -597.496} C_VEL
LIN {X 0,Y 601.548,Z 390.685,A -85,B 0,C 180,E1 -597.938,E2 -597.938} C_VEL
LIN {X 0,Y 601.5,Z 401.609,A -85,B 0,C 180,E1 -598.439,E2 -598.439} C_VEL
LIN {X 0,Y 601.453,Z 412.315,A -85,B 0,C 180,E1 -599.061,E2 -599.061} C_VEL
LIN {X 0,Y 601.452,Z 423.832,A -85,B 0,C 180,E1 -599.903,E2 -599.903} C_VEL
LIN {X 0,Y 601.438,Z 431.651,A -85,B 0,C 180,E1 -600.609,E2 -600.609} C_VEL
LIN {X 0,Y 601.389,Z 438.926,A -85,B 0,C 180,E1 -601.372,E2 -601.372} C_VEL
LIN {X 0,Y 601.384,Z 447.041,A -85,B 0,C 180,E1 -602.415,E2 -602.415} C_VEL
LIN {X 0,Y 601.348,Z 453.429,A -85,B 0,C 180,E1 -603.448,E2 -603.448} C_VEL
LIN {X 0,Y 601.336,Z 458.065,A -85,B 0,C 180,E1 -604.38,E2 -604.38} C_VEL
LIN {X 0,Y 601.353,Z 461.032,A -85,B 0,C 180,E1 -605.121,E2 -605.121} C_VEL
LIN {X 0,Y 601.348,Z 463.459,A -85,B 0,C 180,E1 -605.856,E2 -605.856} C_VEL
LIN {X 0,Y 601.32,Z 465.298,A -85,B 0,C 180,E1 -606.587,E2 -606.587} C_VEL
LIN {X 0,Y 601.343,Z 466.799,A -85,B 0,C 180,E1 -607.399,E2 -607.399} C_VEL
LIN {X 0,Y 601.332,Z 467.549,A -85,B 0,C 180,E1 -608.039,E2 -608.039} C_VEL
LIN {X 0,Y 601.351,Z 467.968,A -85,B 0,C 180,E1 -609.208,E2 -609.208} C_VEL
LIN {X 0,Y 601.314,Z 467.412,A -85,B 0,C 180,E1 -610.189,E2 -610.189} C_VEL
LIN {X 0,Y 601.342,Z 465.968,A -85,B 0,C 180,E1 -611.188,E2 -611.188} C_VEL
LIN {X 0,Y 601.335,Z 462.114,A -85,B 0,C 180,E1 -612.662,E2 -612.662} C_VEL
LIN {X 0,Y 601.36,Z 458.057,A -85,B 0,C 180,E1 -613.712,E2 -613.712} C_VEL
LIN {X 0,Y 601.36,Z 451.787,A -85,B 0,C 180,E1 -614.929,E2 -614.929} C_VEL
LIN {X 0,Y 601.391,Z 444.658,A -85,B 0,C 180,E1 -616.003,E2 -616.003} C_VEL
LIN {X 0,Y 601.415,Z 436.415,A -85,B 0,C 180,E1 -617.001,E2 -617.001} C_VEL
LIN {X 0,Y 601.431,Z 427.664,A -85,B 0,C 180,E1 -617.859,E2 -617.859} C_VEL
LIN {X 0,Y 601.468,Z 416.59,A -85,B 0,C 180,E1 -618.739,E2 -618.739} C_VEL
LIN {X 0,Y 601.485,Z 406.286,A -85,B 0,C 180,E1 -619.397,E2 -619.397} C_VEL
LIN {X 0,Y 601.556,Z 394.383,A -85,B 0,C 180,E1 -619.993,E2 -619.993} C_VEL
LIN {X 0,Y 601.573,Z 382.094,A -85,B 0,C 180,E1 -620.46,E2 -620.46} C_VEL
LIN {X 0,Y 601.616,Z 369.45,A -85,B 0,C 180,E1 -620.8,E2 -620.8} C_VEL
LIN {X 0,Y 601.627,Z 356.29,A -85,B 0,C 180,E1 -621.012,E2 -621.012} C_VEL
LIN {X 0,Y 601.458,Z 257.549,A -85,B 0,C 180,E1 -622.204,E2 -622.204} C_VEL
LIN {X 0,Y 601.387,Z 256.381,A -85,B 0,C 180,E1 -622.291,E2 -622.291} C_VEL
LIN {X 0,Y 601.487,Z 238.178,A -85,B 0,C 180,E1 -625.142,E2 -625.142} C_VEL
LIN {X 0,Y 601.529,Z 220.285,A -85,B 0,C 180,E1 -627.992,E2 -627.992} C_VEL
LIN {X 0,Y 601.457,Z 212.174,A -85,B 0,C 180,E1 -629.332,E2 -629.332} C_VEL
LIN {X 0,Y 601.367,Z 212.07,A -85,B 0,C 180,E1 -632.01,E2 -632.01} C_VEL
LIN {X 0,Y 601.351,Z 212.073,A -85,B 0,C 180,E1 -634.022,E2 -634.022} C_VEL
LIN {X 0,Y 601.36,Z 212.072,A -85,B 0,C 180,E1 -636.039,E2 -636.039} C_VEL
LIN {X 0,Y 601.393,Z 212.068,A -85,B 0,C 180,E1 -638.062,E2 -638.062} C_VEL
LIN {X 0,Y 601.358,Z 212.07,A -85,B 0,C 180,E1 -640.778,E2 -640.778} C_VEL
LIN {X 0,Y 601.383,Z 212.076,A -85,B 0,C 180,E1 -643.518,E2 -643.518} C_VEL
LIN {X 0,Y 601.378,Z 212.07,A -85,B 0,C 180,E1 -646.29,E2 -646.29} C_VEL
LIN {X 0,Y 601.371,Z 212.069,A -85,B 0,C 180,E1 -649.101,E2 -649.101} C_VEL
LIN {X 0,Y 601.372,Z 212.08,A -85,B 0,C 180,E1 -651.962,E2 -651.962} C_VEL
LIN {X 0,Y 601.414,Z 212.069,A -85,B 0,C 180,E1 -654.299,E2 -654.299} C_VEL
LIN {X 0,Y 601.346,Z 212.071,A -85,B 0,C 180,E1 -657.117,E2 -657.117} C_VEL
LIN {X 0,Y 601.356,Z 212.071,A -85,B 0,C 180,E1 -659.397,E2 -659.397} C_VEL
LIN {X 0,Y 601.366,Z 212.072,A -85,B 0,C 180,E1 -661.73,E2 -661.73} C_VEL
LIN {X 0,Y 601.376,Z 212.075,A -85,B 0,C 180,E1 -664.123,E2 -664.123} C_VEL
LIN {X 0,Y 601.356,Z 212.079,A -85,B 0,C 180,E1 -666.587,E2 -666.587} C_VEL
LIN {X 0,Y 601.353,Z 212.072,A -85,B 0,C 180,E1 -669.132,E2 -669.132} C_VEL
LIN {X 0,Y 601.372,Z 212.069,A -85,B 0,C 180,E1 -671.771,E2 -671.771} C_VEL
LIN {X 0,Y 601.371,Z 212.077,A -85,B 0,C 180,E1 -674.536,E2 -674.536} C_VEL
LIN {X 0,Y 601.405,Z 212.07,A -85,B 0,C 180,E1 -676.431,E2 -676.431} C_VEL
LIN {X 0,Y 601.384,Z 212.069,A -85,B 0,C 180,E1 -679.431,E2 -679.431} C_VEL
LIN {X 0,Y 601.362,Z 212.07,A -85,B 0,C 180,E1 -681.733,E2 -681.733} C_VEL
LIN {X 0,Y 601.353,Z 212.071,A -85,B 0,C 180,E1 -684.248,E2 -684.248} C_VEL
LIN {X 0,Y 601.376,Z 212.072,A -85,B 0,C 180,E1 -686.688,E2 -686.688} C_VEL
LIN {X 0,Y 601.386,Z 212.077,A -85,B 0,C 180,E1 -689.06,E2 -689.06} C_VEL
LIN {X 0,Y 601.425,Z 212.07,A -85,B 0,C 180,E1 -691.377,E2 -691.377} C_VEL
LIN {X 0,Y 601.365,Z 212.069,A -85,B 0,C 180,E1 -694.144,E2 -694.144} C_VEL
LIN {X 0,Y 601.358,Z 212.07,A -85,B 0,C 180,E1 -696.591,E2 -696.591} C_VEL
LIN {X 0,Y 601.423,Z 212.074,A -85,B 0,C 180,E1 -699.482,E2 -699.482} C_VEL
LIN {X 0,Y 601.36,Z 212.071,A -85,B 0,C 180,E1 -702.314,E2 -702.314} C_VEL
LIN {X 0,Y 601.378,Z 212.068,A -85,B 0,C 180,E1 -704.411,E2 -704.411} C_VEL
LIN {X 0,Y 601.384,Z 212.067,A -85,B 0,C 180,E1 -706.487,E2 -706.487} C_VEL
LIN {X 0,Y 601.351,Z 212.072,A -85,B 0,C 180,E1 -709.027,E2 -709.027} C_VEL
LIN {X 0,Y 601.382,Z 212.069,A -85,B 0,C 180,E1 -711.265,E2 -711.265} C_VEL
LIN {X 0,Y 601.41,Z 212.076,A -85,B 0,C 180,E1 -713.966,E2 -713.966} C_VEL
LIN {X 0,Y 601.379,Z 212.069,A -85,B 0,C 180,E1 -716.653,E2 -716.653} C_VEL
LIN {X 0,Y 601.407,Z 212.066,A -85,B 0,C 180,E1 -718.663,E2 -718.663} C_VEL
LIN {X 0,Y 601.443,Z 212.063,A -85,B 0,C 180,E1 -720.672,E2 -720.672} C_VEL
LIN {X 0,Y 601.361,Z 212.07,A -85,B 0,C 180,E1 -723.352,E2 -723.352} C_VEL
LIN {X 0,Y 601.391,Z 212.066,A -85,B 0,C 180,E1 -725.367,E2 -725.367} C_VEL
LIN {X 0,Y 601.375,Z 212.068,A -85,B 0,C 180,E1 -727.388,E2 -727.388} C_VEL
LIN {X 0,Y 601.39,Z 212.071,A -85,B 0,C 180,E1 -730.098,E2 -730.098} C_VEL
LIN {X 0,Y 601.415,Z 212.07,A -85,B 0,C 180,E1 -732.83,E2 -732.83} C_VEL
LIN {X 0,Y 601.395,Z 212.065,A -85,B 0,C 180,E1 -735.594,E2 -735.594} C_VEL
LIN {X 0,Y 601.38,Z 212.067,A -85,B 0,C 180,E1 -737.691,E2 -737.691} C_VEL
LIN {X 0,Y 601.388,Z 212.066,A -85,B 0,C 180,E1 -739.812,E2 -739.812} C_VEL
LIN {X 0,Y 601.415,Z 212.069,A -85,B 0,C 180,E1 -742.604,E2 -742.604} C_VEL
LIN {X 0,Y 601.432,Z 212.062,A -85,B 0,C 180,E1 -745.619,E2 -745.619} C_VEL
LIN {X 0,Y 601.374,Z 212.068,A -85,B 0,C 180,E1 -747.871,E2 -747.871} C_VEL
LIN {X 0,Y 601.41,Z 212.063,A -85,B 0,C 180,E1 -750.167,E2 -750.167} C_VEL
LIN {X 0,Y 601.403,Z 212.067,A -85,B 0,C 180,E1 -752.711,E2 -752.711} C_VEL
LIN {X 0,Y 601.383,Z 212.075,A -85,B 0,C 180,E1 -755.109,E2 -755.109} C_VEL
LIN {X 0,Y 601.441,Z 212.071,A -85,B 0,C 180,E1 -757.42,E2 -757.42} C_VEL
LIN {X 0,Y 601.411,Z 212.064,A -85,B 0,C 180,E1 -760.572,E2 -760.572} C_VEL
LIN {X 0,Y 601.38,Z 212.067,A -85,B 0,C 180,E1 -762.674,E2 -762.674} C_VEL
LIN {X 0,Y 601.411,Z 212.072,A -85,B 0,C 180,E1 -765.48,E2 -765.48} C_VEL
LIN {X 0,Y 601.422,Z 212.063,A -85,B 0,C 180,E1 -768.408,E2 -768.408} C_VEL
LIN {X 0,Y 601.398,Z 212.065,A -85,B 0,C 180,E1 -770.871,E2 -770.871} C_VEL
LIN {X 0,Y 601.393,Z 212.069,A -85,B 0,C 180,E1 -773.415,E2 -773.415} C_VEL
LIN {X 0,Y 601.439,Z 212.07,A -85,B 0,C 180,E1 -776.065,E2 -776.065} C_VEL
LIN {X 0,Y 601.408,Z 212.064,A -85,B 0,C 180,E1 -779.056,E2 -779.056} C_VEL
LIN {X 0,Y 601.413,Z 212.064,A -85,B 0,C 180,E1 -781.371,E2 -781.371} C_VEL
LIN {X 0,Y 601.399,Z 212.067,A -85,B 0,C 180,E1 -783.635,E2 -783.635} C_VEL
LIN {X 0,Y 601.421,Z 212.067,A -85,B 0,C 180,E1 -785.857,E2 -785.857} C_VEL
LIN {X 0,Y 601.452,Z 212.238,A -85,B 0,C 180,E1 -788.222,E2 -788.222} C_VEL
LIN {X 0,Y 601.612,Z 218.34,A -85,B 0,C 180,E1 -789.158,E2 -789.158} C_VEL
LIN {X 0,Y 601.53,Z 237.431,A -85,B 0,C 180,E1 -791.963,E2 -791.963} C_VEL
LIN {X 0,Y 601.45,Z 255.53,A -85,B 0,C 180,E1 -794.582,E2 -794.582} C_VEL
LIN {X 0,Y 601.461,Z 271.271,A -85,B 0,C 180,E1 -796.807,E2 -796.807} C_VEL
LIN {X 0,Y 601.67,Z 274.64,A -85,B 0,C 180,E1 -796.876,E2 -796.876} C_VEL
LIN {X 0,Y 601.62,Z 378.895,A -85,B 0,C 180,E1 -798.139,E2 -798.139} C_VEL
LIN {X 0,Y 601.592,Z 392.183,A -85,B 0,C 180,E1 -798.437,E2 -798.437} C_VEL
LIN {X 0,Y 601.551,Z 403.914,A -85,B 0,C 180,E1 -798.826,E2 -798.826} C_VEL
LIN {X 0,Y 601.531,Z 414.904,A -85,B 0,C 180,E1 -799.31,E2 -799.31} C_VEL
LIN {X 0,Y 601.462,Z 425.565,A -85,B 0,C 180,E1 -799.905,E2 -799.905} C_VEL
LIN {X 0,Y 601.447,Z 436.464,A -85,B 0,C 180,E1 -800.668,E2 -800.668} C_VEL
LIN {X 0,Y 601.424,Z 445.309,A -85,B 0,C 180,E1 -801.431,E2 -801.431} C_VEL
LIN {X 0,Y 601.397,Z 453.469,A -85,B 0,C 180,E1 -802.276,E2 -802.276} C_VEL
LIN {X 0,Y 601.383,Z 461.463,A -85,B 0,C 180,E1 -803.288,E2 -803.288} C_VEL
LIN {X 0,Y 601.372,Z 467.861,A -85,B 0,C 180,E1 -804.298,E2 -804.298} C_VEL
LIN {X 0,Y 601.336,Z 472.946,A -85,B 0,C 180,E1 -805.306,E2 -805.306} C_VEL
LIN {X 0,Y 601.367,Z 476.893,A -85,B 0,C 180,E1 -806.314,E2 -806.314} C_VEL
LIN {X 0,Y 601.325,Z 479.806,A -85,B 0,C 180,E1 -807.319,E2 -807.319} C_VEL
LIN {X 0,Y 601.341,Z 481.2,A -85,B 0,C 180,E1 -807.99,E2 -807.99} C_VEL
LIN {X 0,Y 601.339,Z 482.783,A -85,B 0,C 180,E1 -809.329,E2 -809.329} C_VEL
LIN {X 0,Y 601.335,Z 483,A -85,B 0,C 180,E1 -809.999,E2 -809.999} C_VEL
LIN {X 0,Y 601.347,Z 482.186,A -85,B 0,C 180,E1 -811.338,E2 -811.338} C_VEL
LIN {X 0,Y 601.341,Z 481.204,A -85,B 0,C 180,E1 -812.008,E2 -812.008} C_VEL
LIN {X 0,Y 601.325,Z 479.812,A -85,B 0,C 180,E1 -812.678,E2 -812.678} C_VEL
LIN {X 0,Y 601.367,Z 476.9,A -85,B 0,C 180,E1 -813.684,E2 -813.684} C_VEL
LIN {X 0,Y 601.336,Z 472.954,A -85,B 0,C 180,E1 -814.692,E2 -814.692} C_VEL
LIN {X 0,Y 601.372,Z 466.884,A -85,B 0,C 180,E1 -815.868,E2 -815.868} C_VEL
LIN {X 0,Y 601.381,Z 460.244,A -85,B 0,C 180,E1 -816.879,E2 -816.879} C_VEL
LIN {X 0,Y 601.4,Z 451.999,A -85,B 0,C 180,E1 -817.891,E2 -817.891} C_VEL
LIN {X 0,Y 601.434,Z 441.612,A -85,B 0,C 180,E1 -818.906,E2 -818.906} C_VEL
LIN {X 0,Y 601.472,Z 430.764,A -85,B 0,C 180,E1 -819.753,E2 -819.753} C_VEL
LIN {X 0,Y 601.495,Z 419.797,A -85,B 0,C 180,E1 -820.433,E2 -820.433} C_VEL
LIN {X 0,Y 601.551,Z 407.669,A -85,B 0,C 180,E1 -821.022,E2 -821.022} C_VEL
LIN {X 0,Y 601.578,Z 395.912,A -85,B 0,C 180,E1 -821.454,E2 -821.454} C_VEL
LIN {X 0,Y 601.608,Z 383.572,A -85,B 0,C 180,E1 -821.774,E2 -821.774} C_VEL
LIN {X 0,Y 601.642,Z 367.83,A -85,B 0,C 180,E1 -822.008,E2 -822.008} C_VEL
LIN {X 0,Y 601.574,Z 272.279,A -85,B 0,C 180,E1 -823.156,E2 -823.156} C_VEL
LIN {X 0,Y 601.453,Z 271.017,A -85,B 0,C 180,E1 -823.213,E2 -823.213} C_VEL
LIN {X 0,Y 601.485,Z 251.925,A -85,B 0,C 180,E1 -825.936,E2 -825.936} C_VEL
LIN {X 0,Y 601.53,Z 233.427,A -85,B 0,C 180,E1 -828.622,E2 -828.622} C_VEL
LIN {X 0,Y 601.645,Z 214.52,A -85,B 0,C 180,E1 -831.409,E2 -831.409} C_VEL
LIN {X 0,Y 601.436,Z 212.145,A -85,B 0,C 180,E1 -831.822,E2 -831.822} C_VEL
LIN {X 0,Y 601.406,Z 212.067,A -85,B 0,C 180,E1 -834.285,E2 -834.285} C_VEL
LIN {X 0,Y 601.455,Z 212.06,A -85,B 0,C 180,E1 -837.109,E2 -837.109} C_VEL
LIN {X 0,Y 601.402,Z 212.07,A -85,B 0,C 180,E1 -840.164,E2 -840.164} C_VEL
LIN {X 0,Y 601.405,Z 212.065,A -85,B 0,C 180,E1 -842.712,E2 -842.712} C_VEL
LIN {X 0,Y 601.383,Z 212.067,A -85,B 0,C 180,E1 -845.109,E2 -845.109} C_VEL
LIN {X 0,Y 601.431,Z 212.063,A -85,B 0,C 180,E1 -847.418,E2 -847.418} C_VEL
LIN {X 0,Y 601.399,Z 212.074,A -85,B 0,C 180,E1 -849.994,E2 -849.994} C_VEL
LIN {X 0,Y 601.38,Z 212.071,A -85,B 0,C 180,E1 -852.671,E2 -852.671} C_VEL
LIN {X 0,Y 601.395,Z 212.066,A -85,B 0,C 180,E1 -855.478,E2 -855.478} C_VEL
LIN {X 0,Y 601.416,Z 212.074,A -85,B 0,C 180,E1 -858.406,E2 -858.406} C_VEL
LIN {X 0,Y 601.387,Z 212.07,A -85,B 0,C 180,E1 -860.87,E2 -860.87} C_VEL
LIN {X 0,Y 601.378,Z 212.068,A -85,B 0,C 180,E1 -863.414,E2 -863.414} C_VEL
LIN {X 0,Y 601.426,Z 212.065,A -85,B 0,C 180,E1 -866.063,E2 -866.063} C_VEL
LIN {X 0,Y 601.389,Z 212.071,A -85,B 0,C 180,E1 -869.055,E2 -869.055} C_VEL
LIN {X 0,Y 601.389,Z 212.068,A -85,B 0,C 180,E1 -871.369,E2 -871.369} C_VEL
LIN {X 0,Y 601.374,Z 212.068,A -85,B 0,C 180,E1 -873.633,E2 -873.633} C_VEL
LIN {X 0,Y 601.389,Z 212.066,A -85,B 0,C 180,E1 -875.855,E2 -875.855} C_VEL
LIN {X 0,Y 601.389,Z 212.074,A -85,B 0,C 180,E1 -878.758,E2 -878.758} C_VEL
LIN {X 0,Y 601.365,Z 212.071,A -85,B 0,C 180,E1 -881.604,E2 -881.604} C_VEL
LIN {X 0,Y 601.393,Z 212.067,A -85,B 0,C 180,E1 -883.71,E2 -883.71} C_VEL
LIN {X 0,Y 601.383,Z 212.068,A -85,B 0,C 180,E1 -886.481,E2 -886.481} C_VEL
LIN {X 0,Y 601.408,Z 212.076,A -85,B 0,C 180,E1 -889.222,E2 -889.222} C_VEL
LIN {X 0,Y 601.371,Z 212.07,A -85,B 0,C 180,E1 -891.936,E2 -891.936} C_VEL
LIN {X 0,Y 601.355,Z 212.072,A -85,B 0,C 180,E1 -893.96,E2 -893.96} C_VEL
LIN {X 0,Y 601.348,Z 212.073,A -85,B 0,C 180,E1 -895.977,E2 -895.977} C_VEL
LIN {X 0,Y 601.37,Z 212.071,A -85,B 0,C 180,E1 -897.988,E2 -897.988} C_VEL
LIN {X 0,Y 601.396,Z 212.069,A -85,B 0,C 180,E1 -899.997,E2 -899.997} C_VEL
LIN {X 0,Y 601.372,Z 212.068,A -85,B 0,C 180,E1 -902.677,E2 -902.677} C_VEL
LIN {X 0,Y 601.386,Z 212.072,A -85,B 0,C 180,E1 -905.362,E2 -905.362} C_VEL
LIN {X 0,Y 601.416,Z 212.069,A -85,B 0,C 180,E1 -908.058,E2 -908.058} C_VEL
LIN {X 0,Y 601.344,Z 212.072,A -85,B 0,C 180,E1 -910.774,E2 -910.774} C_VEL
LIN {X 0,Y 601.369,Z 212.072,A -85,B 0,C 180,E1 -912.325,E2 -912.325} C_VEL
LIN {X 0,Y 600.674,Z 212.158,A -85,B 0,C 180,E1 -912.884,E2 -912.884} C_VEL
LIN {X 0,Y 597.815,Z 212.521,A -85,B 0,C 180,E1 -913.792,E2 -913.792} C_VEL
LIN {X 0,Y 595.42,Z 212.814,A -85,B 0,C 180,E1 -914.523,E2 -914.523} C_VEL
LIN {X 0,Y 594.396,Z 212.938,A -85,B 0,C 180,E1 -915.087,E2 -915.087} C_VEL
LIN {X 0,Y 594.313,Z 212.949,A -85,B 0,C 180,E1 -915.277,E2 -915.277} C_VEL
LIN {X 0,Y 594.321,Z 212.956,A -85,B 0,C 180,E1 -917.903,E2 -917.903} C_VEL
LIN {X 0,Y 594.374,Z 212.942,A -85,B 0,C 180,E1 -920.773,E2 -920.773} C_VEL
LIN {X 0,Y 594.351,Z 212.946,A -85,B 0,C 180,E1 -923.702,E2 -923.702} C_VEL
LIN {X 0,Y 594.346,Z 212.948,A -85,B 0,C 180,E1 -926.697,E2 -926.697} C_VEL
LIN {X 0,Y 594.358,Z 212.943,A -85,B 0,C 180,E1 -928.995,E2 -928.995} C_VEL
LIN {X 0,Y 594.346,Z 212.944,A -85,B 0,C 180,E1 -931.641,E2 -931.641} C_VEL
LIN {X 0,Y 594.375,Z 212.95,A -85,B 0,C 180,E1 -934.576,E2 -934.576} C_VEL
LIN {X 0,Y 594.359,Z 212.945,A -85,B 0,C 180,E1 -937.084,E2 -937.084} C_VEL
LIN {X 0,Y 594.344,Z 212.945,A -85,B 0,C 180,E1 -939.773,E2 -939.773} C_VEL
LIN {X 0,Y 594.353,Z 212.948,A -85,B 0,C 180,E1 -942.371,E2 -942.371} C_VEL
LIN {X 0,Y 594.323,Z 212.952,A -85,B 0,C 180,E1 -945.189,E2 -945.189} C_VEL
LIN {X 0,Y 594.355,Z 212.948,A -85,B 0,C 180,E1 -947.625,E2 -947.625} C_VEL
LIN {X 0,Y 594.415,Z 213.091,A -85,B 0,C 180,E1 -948.666,E2 -948.666} C_VEL
LIN {X 0,Y 594.563,Z 219,A -85,B 0,C 180,E1 -949.658,E2 -949.658} C_VEL
LIN {X 0,Y 594.432,Z 235.853,A -85,B 0,C 180,E1 -952.379,E2 -952.379} C_VEL
LIN {X 0,Y 594.398,Z 253.775,A -85,B 0,C 180,E1 -955.235,E2 -955.235} C_VEL
LIN {X 0,Y 594.431,Z 256.946,A -85,B 0,C 180,E1 -955.7,E2 -955.7} C_VEL
LIN {X 0,Y 594.731,Z 260.128,A -85,B 0,C 180,E1 -955.771,E2 -955.771} C_VEL
LIN {X 0,Y 594.669,Z 364.519,A -85,B 0,C 180,E1 -957.055,E2 -957.055} C_VEL
LIN {X 0,Y 594.658,Z 378.074,A -85,B 0,C 180,E1 -957.371,E2 -957.371} C_VEL
LIN {X 0,Y 594.563,Z 390.933,A -85,B 0,C 180,E1 -957.816,E2 -957.816} C_VEL
LIN {X 0,Y 594.514,Z 401.865,A -85,B 0,C 180,E1 -958.327,E2 -958.327} C_VEL
LIN {X 0,Y 594.456,Z 412.472,A -85,B 0,C 180,E1 -958.953,E2 -958.953} C_VEL
LIN {X 0,Y 594.421,Z 422.944,A -85,B 0,C 180,E1 -959.722,E2 -959.722} C_VEL
LIN {X 0,Y 594.392,Z 430.797,A -85,B 0,C 180,E1 -960.421,E2 -960.421} C_VEL
LIN {X 0,Y 594.332,Z 439.848,A -85,B 0,C 180,E1 -961.387,E2 -961.387} C_VEL
LIN {X 0,Y 594.293,Z 447.992,A -85,B 0,C 180,E1 -962.481,E2 -962.481} C_VEL
LIN {X 0,Y 594.279,Z 454.984,A -85,B 0,C 180,E1 -963.673,E2 -963.673} C_VEL
LIN {X 0,Y 594.286,Z 460.05,A -85,B 0,C 180,E1 -964.804,E2 -964.804} C_VEL
LIN {X 0,Y 594.241,Z 462.743,A -85,B 0,C 180,E1 -965.586,E2 -965.586} C_VEL
LIN {X 0,Y 594.222,Z 464.7,A -85,B 0,C 180,E1 -966.29,E2 -966.29} C_VEL
LIN {X 0,Y 594.248,Z 466.637,A -85,B 0,C 180,E1 -967.28,E2 -967.28} C_VEL
LIN {X 0,Y 594.218,Z 467.868,A -85,B 0,C 180,E1 -968.492,E2 -968.492} C_VEL
LIN {X 0,Y 594.264,Z 467.966,A -85,B 0,C 180,E1 -969.221,E2 -969.221} C_VEL
LIN {X 0,Y 594.214,Z 467.634,A -85,B 0,C 180,E1 -969.942,E2 -969.942} C_VEL
LIN {X 0,Y 594.234,Z 466.168,A -85,B 0,C 180,E1 -971.098,E2 -971.098} C_VEL
LIN {X 0,Y 594.26,Z 462.913,A -85,B 0,C 180,E1 -972.449,E2 -972.449} C_VEL
LIN {X 0,Y 594.263,Z 459.127,A -85,B 0,C 180,E1 -973.512,E2 -973.512} C_VEL
LIN {X 0,Y 594.272,Z 454.171,A -85,B 0,C 180,E1 -974.57,E2 -974.57} C_VEL
LIN {X 0,Y 594.288,Z 447.911,A -85,B 0,C 180,E1 -975.622,E2 -975.622} C_VEL
LIN {X 0,Y 594.34,Z 440.128,A -85,B 0,C 180,E1 -976.67,E2 -976.67} C_VEL
LIN {X 0,Y 594.367,Z 432.088,A -85,B 0,C 180,E1 -977.539,E2 -977.539} C_VEL
LIN {X 0,Y 594.427,Z 423.541,A -85,B 0,C 180,E1 -978.32,E2 -978.32} C_VEL
LIN {X 0,Y 594.454,Z 413.058,A -85,B 0,C 180,E1 -979.097,E2 -979.097} C_VEL
LIN {X 0,Y 594.502,Z 401.415,A -85,B 0,C 180,E1 -979.787,E2 -979.787} C_VEL
LIN {X 0,Y 594.571,Z 389.046,A -85,B 0,C 180,E1 -980.347,E2 -980.347} C_VEL
LIN {X 0,Y 594.609,Z 376.084,A -85,B 0,C 180,E1 -980.777,E2 -980.777} C_VEL
LIN {X 0,Y 594.685,Z 363.333,A -85,B 0,C 180,E1 -981.056,E2 -981.056} C_VEL
LIN {X 0,Y 594.53,Z 258.152,A -85,B 0,C 180,E1 -982.348,E2 -982.348} C_VEL
LIN {X 0,Y 594.373,Z 256.598,A -85,B 0,C 180,E1 -982.421,E2 -982.421} C_VEL
LIN {X 0,Y 594.449,Z 238.7,A -85,B 0,C 180,E1 -985.254,E2 -985.254} C_VEL
LIN {X 0,Y 594.505,Z 222.904,A -85,B 0,C 180,E1 -987.799,E2 -987.799} C_VEL
LIN {X 0,Y 594.48,Z 213.574,A -85,B 0,C 180,E1 -989.324,E2 -989.324} C_VEL
LIN {X 0,Y 594.387,Z 212.993,A -85,B 0,C 180,E1 -989.493,E2 -989.493} C_VEL
LIN {X 0,Y 594.338,Z 212.946,A -85,B 0,C 180,E1 -992.034,E2 -992.034} C_VEL
LIN {X 0,Y 594.348,Z 212.945,A -85,B 0,C 180,E1 -994.749,E2 -994.749} C_VEL
LIN {X 0,Y 594.382,Z 212.951,A -85,B 0,C 180,E1 -997.474,E2 -997.474} C_VEL
LIN {X 0,Y 594.343,Z 212.945,A -85,B 0,C 180,E1 -1000.218,E2 -1000.218} C_VEL
LIN {X 0,Y 594.316,Z 212.949,A -85,B 0,C 180,E1 -1002.985,E2 -1002.985} C_VEL
LIN {X 0,Y 594.326,Z 212.957,A -85,B 0,C 180,E1 -1005.783,E2 -1005.783} C_VEL
LIN {X 0,Y 594.334,Z 212.945,A -85,B 0,C 180,E1 -1008.62,E2 -1008.62} C_VEL
LIN {X 0,Y 594.321,Z 212.951,A -85,B 0,C 180,E1 -1011.506,E2 -1011.506} C_VEL
LIN {X 0,Y 594.351,Z 212.947,A -85,B 0,C 180,E1 -1014.449,E2 -1014.449} C_VEL
LIN {X 0,Y 594.313,Z 212.95,A -85,B 0,C 180,E1 -1016.704,E2 -1016.704} C_VEL
LIN {X 0,Y 594.336,Z 212.945,A -85,B 0,C 180,E1 -1019.002,E2 -1019.002} C_VEL
LIN {X 0,Y 594.338,Z 212.946,A -85,B 0,C 180,E1 -1021.645,E2 -1021.645} C_VEL
LIN {X 0,Y 594.33,Z 212.953,A -85,B 0,C 180,E1 -1024.139,E2 -1024.139} C_VEL
LIN {X 0,Y 594.296,Z 212.951,A -85,B 0,C 180,E1 -1027.094,E2 -1027.094} C_VEL
LIN {X 0,Y 594.311,Z 212.949,A -85,B 0,C 180,E1 -1029.774,E2 -1029.774} C_VEL
LIN {X 0,Y 594.333,Z 212.952,A -85,B 0,C 180,E1 -1032.379,E2 -1032.379} C_VEL
LIN {X 0,Y 594.31,Z 212.951,A -85,B 0,C 180,E1 -1035.197,E2 -1035.197} C_VEL
LIN {X 0,Y 594.312,Z 212.948,A -85,B 0,C 180,E1 -1037.625,E2 -1037.625} C_VEL
LIN {X 0,Y 594.338,Z 212.947,A -85,B 0,C 180,E1 -1040.322,E2 -1040.322} C_VEL
LIN {X 0,Y 594.363,Z 212.953,A -85,B 0,C 180,E1 -1042.917,E2 -1042.917} C_VEL
LIN {X 0,Y 594.345,Z 212.944,A -85,B 0,C 180,E1 -1045.868,E2 -1045.868} C_VEL
LIN {X 0,Y 594.344,Z 212.947,A -85,B 0,C 180,E1 -1048.653,E2 -1048.653} C_VEL
LIN {X 0,Y 594.369,Z 212.949,A -85,B 0,C 180,E1 -1051.046,E2 -1051.046} C_VEL
LIN {X 0,Y 594.327,Z 212.947,A -85,B 0,C 180,E1 -1054.058,E2 -1054.058} C_VEL
LIN {X 0,Y 594.344,Z 212.944,A -85,B 0,C 180,E1 -1056.298,E2 -1056.298} C_VEL
LIN {X 0,Y 594.395,Z 212.944,A -85,B 0,C 180,E1 -1059.228,E2 -1059.228} C_VEL
LIN {X 0,Y 594.324,Z 212.949,A -85,B 0,C 180,E1 -1062.098,E2 -1062.098} C_VEL
LIN {X 0,Y 594.336,Z 212.947,A -85,B 0,C 180,E1 -1064.222,E2 -1064.222} C_VEL
LIN {X 0,Y 594.358,Z 212.944,A -85,B 0,C 180,E1 -1066.324,E2 -1066.324} C_VEL
LIN {X 0,Y 594.33,Z 212.946,A -85,B 0,C 180,E1 -1068.959,E2 -1068.959} C_VEL
LIN {X 0,Y 594.377,Z 212.951,A -85,B 0,C 180,E1 -1071.846,E2 -1071.846} C_VEL
LIN {X 0,Y 594.367,Z 212.943,A -85,B 0,C 180,E1 -1074.575,E2 -1074.575} C_VEL
LIN {X 0,Y 594.368,Z 212.941,A -85,B 0,C 180,E1 -1077.292,E2 -1077.292} C_VEL
LIN {X 0,Y 594.408,Z 212.944,A -85,B 0,C 180,E1 -1080.003,E2 -1080.003} C_VEL
LIN {X 0,Y 594.404,Z 212.94,A -85,B 0,C 180,E1 -1082.713,E2 -1082.713} C_VEL
LIN {X 0,Y 594.358,Z 212.942,A -85,B 0,C 180,E1 -1085.43,E2 -1085.43} C_VEL
LIN {X 0,Y 594.354,Z 212.949,A -85,B 0,C 180,E1 -1088.16,E2 -1088.16} C_VEL
LIN {X 0,Y 594.399,Z 212.939,A -85,B 0,C 180,E1 -1091.075,E2 -1091.075} C_VEL
LIN {X 0,Y 594.37,Z 212.944,A -85,B 0,C 180,E1 -1094.164,E2 -1094.164} C_VEL
LIN {X 0,Y 594.379,Z 212.943,A -85,B 0,C 180,E1 -1097.196,E2 -1097.196} C_VEL
LIN {X 0,Y 594.361,Z 212.942,A -85,B 0,C 180,E1 -1100.056,E2 -1100.056} C_VEL
LIN {X 0,Y 594.359,Z 212.953,A -85,B 0,C 180,E1 -1102.969,E2 -1102.969} C_VEL
LIN {X 0,Y 594.351,Z 212.943,A -85,B 0,C 180,E1 -1105.947,E2 -1105.947} C_VEL
LIN {X 0,Y 594.331,Z 212.946,A -85,B 0,C 180,E1 -1108.231,E2 -1108.231} C_VEL
LIN {X 0,Y 594.373,Z 212.942,A -85,B 0,C 180,E1 -1110.562,E2 -1110.562} C_VEL
LIN {X 0,Y 594.382,Z 212.945,A -85,B 0,C 180,E1 -1112.952,E2 -1112.952} C_VEL
LIN {X 0,Y 594.334,Z 212.955,A -85,B 0,C 180,E1 -1115.412,E2 -1115.412} C_VEL
LIN {X 0,Y 594.385,Z 212.941,A -85,B 0,C 180,E1 -1117.942,E2 -1117.942} C_VEL
LIN {X 0,Y 594.371,Z 212.942,A -85,B 0,C 180,E1 -1120.82,E2 -1120.82} C_VEL
LIN {X 0,Y 594.353,Z 212.949,A -85,B 0,C 180,E1 -1123.302,E2 -1123.302} C_VEL
LIN {X 0,Y 594.355,Z 212.945,A -85,B 0,C 180,E1 -1126.163,E2 -1126.163} C_VEL
LIN {X 0,Y 594.379,Z 212.94,A -85,B 0,C 180,E1 -1128.535,E2 -1128.535} C_VEL
LIN {X 0,Y 594.376,Z 212.942,A -85,B 0,C 180,E1 -1131.298,E2 -1131.298} C_VEL
LIN {X 0,Y 594.354,Z 212.951,A -85,B 0,C 180,E1 -1133.755,E2 -1133.755} C_VEL
LIN {X 0,Y 594.382,Z 212.946,A -85,B 0,C 180,E1 -1136.238,E2 -1136.238} C_VEL
LIN {X 0,Y 594.374,Z 212.942,A -85,B 0,C 180,E1 -1138.649,E2 -1138.649} C_VEL
LIN {X 0,Y 594.383,Z 212.939,A -85,B 0,C 180,E1 -1141.044,E2 -1141.044} C_VEL
LIN {X 0,Y 594.387,Z 212.939,A -85,B 0,C 180,E1 -1143.3,E2 -1143.3} C_VEL
LIN {X 0,Y 594.356,Z 212.944,A -85,B 0,C 180,E1 -1145.575,E2 -1145.575} C_VEL
LIN {X 0,Y 594.396,Z 213.132,A -85,B 0,C 180,E1 -1148.087,E2 -1148.087} C_VEL
LIN {X 0,Y 594.695,Z 216.838,A -85,B 0,C 180,E1 -1148.678,E2 -1148.678} C_VEL
LIN {X 0,Y 594.574,Z 236.224,A -85,B 0,C 180,E1 -1151.566,E2 -1151.566} C_VEL
LIN {X 0,Y 594.486,Z 254.323,A -85,B 0,C 180,E1 -1154.221,E2 -1154.221} C_VEL
LIN {X 0,Y 594.43,Z 271.264,A -85,B 0,C 180,E1 -1156.648,E2 -1156.648} C_VEL
LIN {X 0,Y 594.769,Z 274.64,A -85,B 0,C 180,E1 -1156.721,E2 -1156.721} C_VEL
LIN {X 0,Y 594.674,Z 378.895,A -85,B 0,C 180,E1 -1157.998,E2 -1157.998} C_VEL
LIN {X 0,Y 594.641,Z 392.184,A -85,B 0,C 180,E1 -1158.3,E2 -1158.3} C_VEL
LIN {X 0,Y 594.589,Z 405.364,A -85,B 0,C 180,E1 -1158.749,E2 -1158.749} C_VEL
LIN {X 0,Y 594.538,Z 416.614,A -85,B 0,C 180,E1 -1159.269,E2 -1159.269} C_VEL
LIN {X 0,Y 594.455,Z 428.186,A -85,B 0,C 180,E1 -1159.956,E2 -1159.956} C_VEL
LIN {X 0,Y 594.414,Z 438.585,A -85,B 0,C 180,E1 -1160.729,E2 -1160.729} C_VEL
LIN {X 0,Y 594.349,Z 447.022,A -85,B 0,C 180,E1 -1161.499,E2 -1161.499} C_VEL
LIN {X 0,Y 594.348,Z 454.952,A -85,B 0,C 180,E1 -1162.354,E2 -1162.354} C_VEL
LIN {X 0,Y 594.282,Z 462.825,A -85,B 0,C 180,E1 -1163.41,E2 -1163.41} C_VEL
LIN {X 0,Y 594.289,Z 469.675,A -85,B 0,C 180,E1 -1164.57,E2 -1164.57} C_VEL
LIN {X 0,Y 594.27,Z 474.367,A -85,B 0,C 180,E1 -1165.59,E2 -1165.59} C_VEL
LIN {X 0,Y 594.267,Z 477.953,A -85,B 0,C 180,E1 -1166.609,E2 -1166.609} C_VEL
LIN {X 0,Y 594.226,Z 479.806,A -85,B 0,C 180,E1 -1167.287,E2 -1167.287} C_VEL
LIN {X 0,Y 594.24,Z 481.199,A -85,B 0,C 180,E1 -1167.966,E2 -1167.966} C_VEL
LIN {X 0,Y 594.239,Z 482.783,A -85,B 0,C 180,E1 -1169.321,E2 -1169.321} C_VEL
LIN {X 0,Y 594.236,Z 483,A -85,B 0,C 180,E1 -1169.999,E2 -1169.999} C_VEL
LIN {X 0,Y 594.247,Z 482.186,A -85,B 0,C 180,E1 -1171.354,E2 -1171.354} C_VEL
LIN {X 0,Y 594.24,Z 481.203,A -85,B 0,C 180,E1 -1172.032,E2 -1172.032} C_VEL
LIN {X 0,Y 594.226,Z 479.812,A -85,B 0,C 180,E1 -1172.711,E2 -1172.711} C_VEL
LIN {X 0,Y 594.288,Z 476.9,A -85,B 0,C 180,E1 -1173.728,E2 -1173.728} C_VEL
LIN {X 0,Y 594.241,Z 472.954,A -85,B 0,C 180,E1 -1174.748,E2 -1174.748} C_VEL
LIN {X 0,Y 594.304,Z 466.884,A -85,B 0,C 180,E1 -1175.938,E2 -1175.938} C_VEL
LIN {X 0,Y 594.308,Z 460.244,A -85,B 0,C 180,E1 -1176.961,E2 -1176.961} C_VEL
LIN {X 0,Y 594.359,Z 452,A -85,B 0,C 180,E1 -1177.985,E2 -1177.985} C_VEL
LIN {X 0,Y 594.404,Z 441.613,A -85,B 0,C 180,E1 -1179.012,E2 -1179.012} C_VEL
LIN {X 0,Y 594.444,Z 430.764,A -85,B 0,C 180,E1 -1179.87,E2 -1179.87} C_VEL
LIN {X 0,Y 594.507,Z 419.799,A -85,B 0,C 180,E1 -1180.557,E2 -1180.557} C_VEL
LIN {X 0,Y 594.601,Z 407.167,A -85,B 0,C 180,E1 -1181.175,E2 -1181.175} C_VEL
LIN {X 0,Y 594.62,Z 395.91,A -85,B 0,C 180,E1 -1181.59,E2 -1181.59} C_VEL
LIN {X 0,Y 594.66,Z 383.57,A -85,B 0,C 180,E1 -1181.913,E2 -1181.913} C_VEL
LIN {X 0,Y 594.709,Z 367.83,A -85,B 0,C 180,E1 -1182.15,E2 -1182.15} C_VEL
LIN {X 0,Y 594.637,Z 273.03,A -85,B 0,C 180,E1 -1183.302,E2 -1183.302} C_VEL
LIN {X 0,Y 594.424,Z 271.012,A -85,B 0,C 180,E1 -1183.372,E2 -1183.372} C_VEL
LIN {X 0,Y 594.489,Z 251.925,A -85,B 0,C 180,E1 -1186.129,E2 -1186.129} C_VEL
LIN {X 0,Y 594.593,Z 233.257,A -85,B 0,C 180,E1 -1188.873,E2 -1188.873} C_VEL
LIN {X 0,Y 594.698,Z 215.727,A -85,B 0,C 180,E1 -1191.489,E2 -1191.489} C_VEL
LIN {X 0,Y 594.378,Z 213.027,A -85,B 0,C 180,E1 -1191.957,E2 -1191.957} C_VEL
LIN {X 0,Y 594.367,Z 212.943,A -85,B 0,C 180,E1 -1194.446,E2 -1194.446} C_VEL
LIN {X 0,Y 594.384,Z 212.94,A -85,B 0,C 180,E1 -1196.698,E2 -1196.698} C_VEL
LIN {X 0,Y 594.374,Z 212.941,A -85,B 0,C 180,E1 -1198.997,E2 -1198.997} C_VEL
LIN {X 0,Y 594.389,Z 212.945,A -85,B 0,C 180,E1 -1201.643,E2 -1201.643} C_VEL
LIN {X 0,Y 594.368,Z 212.943,A -85,B 0,C 180,E1 -1204.579,E2 -1204.579} C_VEL
LIN {X 0,Y 594.386,Z 212.942,A -85,B 0,C 180,E1 -1207.607,E2 -1207.607} C_VEL
LIN {X 0,Y 594.36,Z 212.946,A -85,B 0,C 180,E1 -1210.566,E2 -1210.566} C_VEL
LIN {X 0,Y 594.356,Z 212.942,A -85,B 0,C 180,E1 -1213.299,E2 -1213.299} C_VEL
LIN {X 0,Y 594.357,Z 212.951,A -85,B 0,C 180,E1 -1216.16,E2 -1216.16} C_VEL
LIN {X 0,Y 594.372,Z 212.949,A -85,B 0,C 180,E1 -1218.534,E2 -1218.534} C_VEL
LIN {X 0,Y 594.361,Z 212.942,A -85,B 0,C 180,E1 -1221.296,E2 -1221.296} C_VEL
LIN {X 0,Y 594.341,Z 212.945,A -85,B 0,C 180,E1 -1223.753,E2 -1223.753} C_VEL
LIN {X 0,Y 594.372,Z 212.946,A -85,B 0,C 180,E1 -1226.237,E2 -1226.237} C_VEL
LIN {X 0,Y 594.359,Z 212.954,A -85,B 0,C 180,E1 -1228.647,E2 -1228.647} C_VEL
LIN {X 0,Y 594.366,Z 212.947,A -85,B 0,C 180,E1 -1231.042,E2 -1231.042} C_VEL
LIN {X 0,Y 594.358,Z 212.945,A -85,B 0,C 180,E1 -1233.297,E2 -1233.297} C_VEL
LIN {X 0,Y 594.329,Z 212.947,A -85,B 0,C 180,E1 -1235.575,E2 -1235.575} C_VEL
LIN {X 0,Y 594.345,Z 212.948,A -85,B 0,C 180,E1 -1238.494,E2 -1238.494} C_VEL
LIN {X 0,Y 594.351,Z 212.948,A -85,B 0,C 180,E1 -1241.379,E2 -1241.379} C_VEL
LIN {X 0,Y 594.362,Z 212.945,A -85,B 0,C 180,E1 -1243.512,E2 -1243.512} C_VEL
LIN {X 0,Y 594.342,Z 212.945,A -85,B 0,C 180,E1 -1246.318,E2 -1246.318} C_VEL
LIN {X 0,Y 594.367,Z 212.95,A -85,B 0,C 180,E1 -1249.092,E2 -1249.092} C_VEL
LIN {X 0,Y 594.329,Z 212.948,A -85,B 0,C 180,E1 -1251.84,E2 -1251.84} C_VEL
LIN {X 0,Y 594.316,Z 212.95,A -85,B 0,C 180,E1 -1253.888,E2 -1253.888} C_VEL
LIN {X 0,Y 594.306,Z 212.951,A -85,B 0,C 180,E1 -1255.929,E2 -1255.929} C_VEL
LIN {X 0,Y 594.345,Z 212.947,A -85,B 0,C 180,E1 -1257.965,E2 -1257.965} C_VEL
LIN {X 0,Y 594.367,Z 212.944,A -85,B 0,C 180,E1 -1259.997,E2 -1259.997} C_VEL
LIN {X 0,Y 594.344,Z 212.944,A -85,B 0,C 180,E1 -1262.708,E2 -1262.708} C_VEL
LIN {X 0,Y 594.353,Z 212.949,A -85,B 0,C 180,E1 -1265.425,E2 -1265.425} C_VEL
LIN {X 0,Y 594.357,Z 212.946,A -85,B 0,C 180,E1 -1268.155,E2 -1268.155} C_VEL
LIN {X 0,Y 594.342,Z 212.945,A -85,B 0,C 180,E1 -1271.058,E2 -1271.058} C_VEL
LIN {X 0,Y 594.349,Z 212.95,A -85,B 0,C 180,E1 -1273.676,E2 -1273.676} C_VEL
LIN {X 0,Y 594.313,Z 212.949,A -85,B 0,C 180,E1 -1275.277,E2 -1275.277} C_VEL
LIN {X 0,Y 593.649,Z 213.04,A -85,B 0,C 180,E1 -1275.843,E2 -1275.843} C_VEL
LIN {X 0,Y 590.792,Z 213.401,A -85,B 0,C 180,E1 -1276.761,E2 -1276.761} C_VEL
LIN {X 0,Y 588.382,Z 213.702,A -85,B 0,C 180,E1 -1277.499,E2 -1277.499} C_VEL
LIN {X 0,Y 587.354,Z 213.826,A -85,B 0,C 180,E1 -1278.069,E2 -1278.069} C_VEL
LIN {X 0,Y 587.275,Z 213.832,A -85,B 0,C 180,E1 -1278.262,E2 -1278.262} C_VEL
LIN {X 0,Y 587.304,Z 213.821,A -85,B 0,C 180,E1 -1281.035,E2 -1281.035} C_VEL
LIN {X 0,Y 587.289,Z 213.823,A -85,B 0,C 180,E1 -1283.256,E2 -1283.256} C_VEL
LIN {X 0,Y 587.295,Z 213.823,A -85,B 0,C 180,E1 -1285.514,E2 -1285.514} C_VEL
LIN {X 0,Y 587.307,Z 213.824,A -85,B 0,C 180,E1 -1287.816,E2 -1287.816} C_VEL
LIN {X 0,Y 587.305,Z 213.83,A -85,B 0,C 180,E1 -1290.508,E2 -1290.508} C_VEL
LIN {X 0,Y 587.308,Z 213.822,A -85,B 0,C 180,E1 -1293.11,E2 -1293.11} C_VEL
LIN {X 0,Y 587.326,Z 213.82,A -85,B 0,C 180,E1 -1295.893,E2 -1295.893} C_VEL
LIN {X 0,Y 587.303,Z 213.831,A -85,B 0,C 180,E1 -1298.476,E2 -1298.476} C_VEL
LIN {X 0,Y 587.33,Z 213.822,A -85,B 0,C 180,E1 -1301.152,E2 -1301.152} C_VEL
LIN {X 0,Y 587.295,Z 213.824,A -85,B 0,C 180,E1 -1304.112,E2 -1304.112} C_VEL
LIN {X 0,Y 587.304,Z 213.832,A -85,B 0,C 180,E1 -1306.995,E2 -1306.995} C_VEL
LIN {X 0,Y 587.361,Z 214.032,A -85,B 0,C 180,E1 -1308.573,E2 -1308.573} C_VEL
LIN {X 0,Y 587.605,Z 217.118,A -85,B 0,C 180,E1 -1309.108,E2 -1309.108} C_VEL
LIN {X 0,Y 587.454,Z 233.983,A -85,B 0,C 180,E1 -1311.871,E2 -1311.871} C_VEL
LIN {X 0,Y 587.337,Z 251.463,A -85,B 0,C 180,E1 -1314.695,E2 -1314.695} C_VEL
LIN {X 0,Y 587.396,Z 257.012,A -85,B 0,C 180,E1 -1315.542,E2 -1315.542} C_VEL
LIN {X 0,Y 587.834,Z 260.94,A -85,B 0,C 180,E1 -1315.622,E2 -1315.622} C_VEL
LIN {X 0,Y 587.725,Z 364.16,A -85,B 0,C 180,E1 -1316.904,E2 -1316.904} C_VEL
LIN {X 0,Y 587.688,Z 377.155,A -85,B 0,C 180,E1 -1317.204,E2 -1317.204} C_VEL
LIN {X 0,Y 587.624,Z 389.671,A -85,B 0,C 180,E1 -1317.632,E2 -1317.632} C_VEL
LIN {X 0,Y 587.529,Z 401.851,A -85,B 0,C 180,E1 -1318.198,E2 -1318.198} C_VEL
LIN {X 0,Y 587.435,Z 412.613,A -85,B 0,C 180,E1 -1318.841,E2 -1318.841} C_VEL
LIN {X 0,Y 587.383,Z 422.56,A -85,B 0,C 180,E1 -1319.578,E2 -1319.578} C_VEL
LIN {X 0,Y 587.338,Z 431.869,A -85,B 0,C 180,E1 -1320.425,E2 -1320.425} C_VEL
LIN {X 0,Y 587.272,Z 439.306,A -85,B 0,C 180,E1 -1321.231,E2 -1321.231} C_VEL
LIN {X 0,Y 587.248,Z 446.52,A -85,B 0,C 180,E1 -1322.179,E2 -1322.179} C_VEL
LIN {X 0,Y 587.208,Z 453.538,A -85,B 0,C 180,E1 -1323.334,E2 -1323.334} C_VEL
LIN {X 0,Y 587.153,Z 458.932,A -85,B 0,C 180,E1 -1324.476,E2 -1324.476} C_VEL
LIN {X 0,Y 587.158,Z 462.454,A -85,B 0,C 180,E1 -1325.45,E2 -1325.45} C_VEL
LIN {X 0,Y 587.114,Z 465.729,A -85,B 0,C 180,E1 -1326.734,E2 -1326.734} C_VEL
LIN {X 0,Y 587.145,Z 466.962,A -85,B 0,C 180,E1 -1327.48,E2 -1327.48} C_VEL
LIN {X 0,Y 587.133,Z 467.69,A -85,B 0,C 180,E1 -1328.22,E2 -1328.22} C_VEL
LIN {X 0,Y 587.142,Z 467.995,A -85,B 0,C 180,E1 -1328.997,E2 -1328.997} C_VEL
LIN {X 0,Y 587.148,Z 467.812,A -85,B 0,C 180,E1 -1329.69,E2 -1329.69} C_VEL
LIN {X 0,Y 587.14,Z 466.362,A -85,B 0,C 180,E1 -1331.003,E2 -1331.003} C_VEL
LIN {X 0,Y 587.152,Z 463.674,A -85,B 0,C 180,E1 -1332.23,E2 -1332.23} C_VEL
LIN {X 0,Y 587.171,Z 460.159,A -85,B 0,C 180,E1 -1333.307,E2 -1333.307} C_VEL
LIN {X 0,Y 587.186,Z 455.506,A -85,B 0,C 180,E1 -1334.379,E2 -1334.379} C_VEL
LIN {X 0,Y 587.254,Z 449.564,A -85,B 0,C 180,E1 -1335.446,E2 -1335.446} C_VEL
LIN {X 0,Y 587.251,Z 442.15,A -85,B 0,C 180,E1 -1336.506,E2 -1336.506} C_VEL
LIN {X 0,Y 587.31,Z 434.603,A -85,B 0,C 180,E1 -1337.387,E2 -1337.387} C_VEL
LIN {X 0,Y 587.346,Z 425.514,A -85,B 0,C 180,E1 -1338.264,E2 -1338.264} C_VEL
LIN {X 0,Y 587.463,Z 415.48,A -85,B 0,C 180,E1 -1339.053,E2 -1339.053} C_VEL
LIN {X 0,Y 587.516,Z 404.397,A -85,B 0,C 180,E1 -1339.751,E2 -1339.751} C_VEL
LIN {X 0,Y 587.593,Z 392.013,A -85,B 0,C 180,E1 -1340.362,E2 -1340.362} C_VEL
LIN {X 0,Y 587.674,Z 380.219,A -85,B 0,C 180,E1 -1340.797,E2 -1340.797} C_VEL
LIN {X 0,Y 587.762,Z 367.362,A -85,B 0,C 180,E1 -1341.124,E2 -1341.124} C_VEL
LIN {X 0,Y 587.743,Z 349.435,A -85,B 0,C 180,E1 -1341.383,E2 -1341.383} C_VEL
LIN {X 0,Y 587.653,Z 259.011,A -85,B 0,C 180,E1 -1342.496,E2 -1342.496} C_VEL
LIN {X 0,Y 587.349,Z 256.757,A -85,B 0,C 180,E1 -1342.567,E2 -1342.567} C_VEL
LIN {X 0,Y 587.43,Z 239.218,A -85,B 0,C 180,E1 -1345.369,E2 -1345.369} C_VEL
LIN {X 0,Y 587.51,Z 224.473,A -85,B 0,C 180,E1 -1347.773,E2 -1347.773} C_VEL
LIN {X 0,Y 587.541,Z 215.12,A -85,B 0,C 180,E1 -1349.316,E2 -1349.316} C_VEL
LIN {X 0,Y 587.348,Z 213.892,A -85,B 0,C 180,E1 -1349.573,E2 -1349.573} C_VEL
LIN {X 0,Y 587.31,Z 213.822,A -85,B 0,C 180,E1 -1352.058,E2 -1352.058} C_VEL
LIN {X 0,Y 587.321,Z 213.822,A -85,B 0,C 180,E1 -1354.806,E2 -1354.806} C_VEL
LIN {X 0,Y 587.343,Z 213.826,A -85,B 0,C 180,E1 -1357.564,E2 -1357.564} C_VEL
LIN {X 0,Y 587.292,Z 213.823,A -85,B 0,C 180,E1 -1360.342,E2 -1360.342} C_VEL
LIN {X 0,Y 587.27,Z 213.828,A -85,B 0,C 180,E1 -1363.144,E2 -1363.144} C_VEL
LIN {X 0,Y 587.276,Z 213.831,A -85,B 0,C 180,E1 -1365.977,E2 -1365.977} C_VEL
LIN {X 0,Y 587.284,Z 213.829,A -85,B 0,C 180,E1 -1368.129,E2 -1368.129} C_VEL
LIN {X 0,Y 587.281,Z 213.828,A -85,B 0,C 180,E1 -1370.308,E2 -1370.308} C_VEL
LIN {X 0,Y 587.278,Z 213.825,A -85,B 0,C 180,E1 -1373.262,E2 -1373.262} C_VEL
LIN {X 0,Y 587.286,Z 213.826,A -85,B 0,C 180,E1 -1375.52,E2 -1375.52} C_VEL
LIN {X 0,Y 587.28,Z 213.827,A -85,B 0,C 180,E1 -1378.6,E2 -1378.6} C_VEL
LIN {X 0,Y 587.29,Z 213.823,A -85,B 0,C 180,E1 -1380.97,E2 -1380.97} C_VEL
LIN {X 0,Y 587.287,Z 213.823,A -85,B 0,C 180,E1 -1383.401,E2 -1383.401} C_VEL
LIN {X 0,Y 587.245,Z 213.831,A -85,B 0,C 180,E1 -1385.904,E2 -1385.904} C_VEL
LIN {X 0,Y 587.281,Z 213.835,A -85,B 0,C 180,E1 -1388.484,E2 -1388.484} C_VEL
LIN {X 0,Y 587.278,Z 213.826,A -85,B 0,C 180,E1 -1391.163,E2 -1391.163} C_VEL
LIN {X 0,Y 587.269,Z 213.826,A -85,B 0,C 180,E1 -1393.957,E2 -1393.957} C_VEL
LIN {X 0,Y 587.277,Z 213.833,A -85,B 0,C 180,E1 -1396.887,E2 -1396.887} C_VEL
LIN {X 0,Y 587.282,Z 213.824,A -85,B 0,C 180,E1 -1399.748,E2 -1399.748} C_VEL
LIN {X 0,Y 587.316,Z 213.822,A -85,B 0,C 180,E1 -1402.395,E2 -1402.395} C_VEL
LIN {X 0,Y 587.306,Z 213.831,A -85,B 0,C 180,E1 -1404.948,E2 -1404.948} C_VEL
LIN {X 0,Y 587.314,Z 213.825,A -85,B 0,C 180,E1 -1407.424,E2 -1407.424} C_VEL
LIN {X 0,Y 587.281,Z 213.825,A -85,B 0,C 180,E1 -1409.831,E2 -1409.831} C_VEL
LIN {X 0,Y 587.285,Z 213.823,A -85,B 0,C 180,E1 -1412.321,E2 -1412.321} C_VEL
LIN {X 0,Y 587.287,Z 213.832,A -85,B 0,C 180,E1 -1415.243,E2 -1415.243} C_VEL
LIN {X 0,Y 587.299,Z 213.822,A -85,B 0,C 180,E1 -1418.229,E2 -1418.229} C_VEL
LIN {X 0,Y 587.329,Z 213.822,A -85,B 0,C 180,E1 -1421.154,E2 -1421.154} C_VEL
LIN {X 0,Y 587.294,Z 213.827,A -85,B 0,C 180,E1 -1424.027,E2 -1424.027} C_VEL
LIN {X 0,Y 587.343,Z 213.819,A -85,B 0,C 180,E1 -1426.157,E2 -1426.157} C_VEL
LIN {X 0,Y 587.289,Z 213.823,A -85,B 0,C 180,E1 -1428.965,E2 -1428.965} C_VEL
LIN {X 0,Y 587.335,Z 213.826,A -85,B 0,C 180,E1 -1431.747,E2 -1431.747} C_VEL
LIN {X 0,Y 587.336,Z 213.819,A -85,B 0,C 180,E1 -1434.51,E2 -1434.51} C_VEL
LIN {X 0,Y 587.337,Z 213.817,A -85,B 0,C 180,E1 -1437.259,E2 -1437.259} C_VEL
LIN {X 0,Y 587.377,Z 213.82,A -85,B 0,C 180,E1 -1440.003,E2 -1440.003} C_VEL
LIN {X 0,Y 587.368,Z 213.816,A -85,B 0,C 180,E1 -1442.746,E2 -1442.746} C_VEL
LIN {X 0,Y 587.326,Z 213.818,A -85,B 0,C 180,E1 -1445.496,E2 -1445.496} C_VEL
LIN {X 0,Y 587.322,Z 213.827,A -85,B 0,C 180,E1 -1448.258,E2 -1448.258} C_VEL
LIN {X 0,Y 587.36,Z 213.816,A -85,B 0,C 180,E1 -1451.136,E2 -1451.136} C_VEL
LIN {X 0,Y 587.331,Z 213.822,A -85,B 0,C 180,E1 -1454.245,E2 -1454.245} C_VEL
LIN {X 0,Y 587.344,Z 213.825,A -85,B 0,C 180,E1 -1456.81,E2 -1456.81} C_VEL
LIN {X 0,Y 587.309,Z 213.821,A -85,B 0,C 180,E1 -1459.578,E2 -1459.578} C_VEL
LIN {X 0,Y 587.317,Z 213.819,A -85,B 0,C 180,E1 -1461.776,E2 -1461.776} C_VEL
LIN {X 0,Y 587.313,Z 213.827,A -85,B 0,C 180,E1 -1464.762,E2 -1464.762} C_VEL
LIN {X 0,Y 587.309,Z 213.822,A -85,B 0,C 180,E1 -1467.684,E2 -1467.684} C_VEL
LIN {X 0,Y 587.322,Z 213.818,A -85,B 0,C 180,E1 -1470.173,E2 -1470.173} C_VEL
LIN {X 0,Y 587.336,Z 213.818,A -85,B 0,C 180,E1 -1472.581,E2 -1472.581} C_VEL
LIN {X 0,Y 587.311,Z 213.827,A -85,B 0,C 180,E1 -1475.058,E2 -1475.058} C_VEL
LIN {X 0,Y 587.342,Z 213.82,A -85,B 0,C 180,E1 -1477.838,E2 -1477.838} C_VEL
LIN {X 0,Y 587.315,Z 213.82,A -85,B 0,C 180,E1 -1480.256,E2 -1480.256} C_VEL
LIN {X 0,Y 587.298,Z 213.825,A -85,B 0,C 180,E1 -1483.115,E2 -1483.115} C_VEL
LIN {X 0,Y 587.31,Z 213.824,A -85,B 0,C 180,E1 -1486.047,E2 -1486.047} C_VEL
LIN {X 0,Y 587.32,Z 213.819,A -85,B 0,C 180,E1 -1488.928,E2 -1488.928} C_VEL
LIN {X 0,Y 587.327,Z 213.824,A -85,B 0,C 180,E1 -1491.519,E2 -1491.519} C_VEL
LIN {X 0,Y 587.289,Z 213.831,A -85,B 0,C 180,E1 -1494.099,E2 -1494.099} C_VEL
LIN {X 0,Y 587.34,Z 213.818,A -85,B 0,C 180,E1 -1496.603,E2 -1496.603} C_VEL
LIN {X 0,Y 587.33,Z 213.818,A -85,B 0,C 180,E1 -1499.032,E2 -1499.032} C_VEL
LIN {X 0,Y 587.319,Z 213.82,A -85,B 0,C 180,E1 -1501.402,E2 -1501.402} C_VEL
LIN {X 0,Y 587.319,Z 213.824,A -85,B 0,C 180,E1 -1503.829,E2 -1503.829} C_VEL
LIN {X 0,Y 587.305,Z 213.828,A -85,B 0,C 180,E1 -1505.991,E2 -1505.991} C_VEL
LIN {X 0,Y 587.36,Z 214.026,A -85,B 0,C 180,E1 -1507.949,E2 -1507.949} C_VEL
LIN {X 0,Y 587.752,Z 218.351,A -85,B 0,C 180,E1 -1508.644,E2 -1508.644} C_VEL
LIN {X 0,Y 587.588,Z 238.637,A -85,B 0,C 180,E1 -1511.7,E2 -1511.7} C_VEL
LIN {X 0,Y 587.453,Z 256.736,A -85,B 0,C 180,E1 -1514.384,E2 -1514.384} C_VEL
LIN {X 0,Y 587.406,Z 271.257,A -85,B 0,C 180,E1 -1516.485,E2 -1516.485} C_VEL
LIN {X 0,Y 587.868,Z 274.64,A -85,B 0,C 180,E1 -1516.562,E2 -1516.562} C_VEL
LIN {X 0,Y 587.751,Z 378.895,A -85,B 0,C 180,E1 -1517.855,E2 -1517.855} C_VEL
LIN {X 0,Y 587.686,Z 392.185,A -85,B 0,C 180,E1 -1518.16,E2 -1518.16} C_VEL
LIN {X 0,Y 587.605,Z 404.765,A -85,B 0,C 180,E1 -1518.59,E2 -1518.59} C_VEL
LIN {X 0,Y 587.555,Z 416.612,A -85,B 0,C 180,E1 -1519.14,E2 -1519.14} C_VEL
LIN {X 0,Y 587.437,Z 428.188,A -85,B 0,C 180,E1 -1519.835,E2 -1519.835} C_VEL
LIN {X 0,Y 587.393,Z 438.586,A -85,B 0,C 180,E1 -1520.617,E2 -1520.617} C_VEL
LIN {X 0,Y 587.3,Z 447.037,A -85,B 0,C 180,E1 -1521.396,E2 -1521.396} C_VEL
LIN {X 0,Y 587.275,Z 454.952,A -85,B 0,C 180,E1 -1522.262,E2 -1522.262} C_VEL
LIN {X 0,Y 587.232,Z 461.462,A -85,B 0,C 180,E1 -1523.125,E2 -1523.125} C_VEL
LIN {X 0,Y 587.236,Z 467.861,A -85,B 0,C 180,E1 -1524.16,E2 -1524.16} C_VEL
LIN {X 0,Y 587.147,Z 472.946,A -85,B 0,C 180,E1 -1525.193,E2 -1525.193} C_VEL
LIN {X 0,Y 587.213,Z 476.892,A -85,B 0,C 180,E1 -1526.225,E2 -1526.225} C_VEL
LIN {X 0,Y 587.132,Z 479.806,A -85,B 0,C 180,E1 -1527.255,E2 -1527.255} C_VEL
LIN {X 0,Y 587.139,Z 481.198,A -85,B 0,C 180,E1 -1527.941,E2 -1527.941} C_VEL
LIN {X 0,Y 587.14,Z 482.784,A -85,B 0,C 180,E1 -1529.313,E2 -1529.313} C_VEL
LIN {X 0,Y 587.137,Z 483,A -85,B 0,C 180,E1 -1529.999,E2 -1529.999} C_VEL
LIN {X 0,Y 587.147,Z 482.187,A -85,B 0,C 180,E1 -1531.371,E2 -1531.371} C_VEL
LIN {X 0,Y 587.139,Z 481.202,A -85,B 0,C 180,E1 -1532.057,E2 -1532.057} C_VEL
LIN {X 0,Y 587.132,Z 479.812,A -85,B 0,C 180,E1 -1532.743,E2 -1532.743} C_VEL
LIN {X 0,Y 587.212,Z 476.899,A -85,B 0,C 180,E1 -1533.773,E2 -1533.773} C_VEL
LIN {X 0,Y 587.147,Z 472.954,A -85,B 0,C 180,E1 -1534.805,E2 -1534.805} C_VEL
LIN {X 0,Y 587.217,Z 466.884,A -85,B 0,C 180,E1 -1536.01,E2 -1536.01} C_VEL
LIN {X 0,Y 587.245,Z 460.245,A -85,B 0,C 180,E1 -1537.045,E2 -1537.045} C_VEL
LIN {X 0,Y 587.297,Z 452,A -85,B 0,C 180,E1 -1538.082,E2 -1538.082} C_VEL
LIN {X 0,Y 587.357,Z 441.614,A -85,B 0,C 180,E1 -1539.121,E2 -1539.121} C_VEL
LIN {X 0,Y 587.44,Z 430.763,A -85,B 0,C 180,E1 -1539.989,E2 -1539.989} C_VEL
LIN {X 0,Y 587.524,Z 419.802,A -85,B 0,C 180,E1 -1540.684,E2 -1540.684} C_VEL
LIN {X 0,Y 587.618,Z 408.21,A -85,B 0,C 180,E1 -1541.263,E2 -1541.263} C_VEL
LIN {X 0,Y 587.685,Z 395.908,A -85,B 0,C 180,E1 -1541.729,E2 -1541.729} C_VEL
LIN {X 0,Y 587.714,Z 383.569,A -85,B 0,C 180,E1 -1542.056,E2 -1542.056} C_VEL
LIN {X 0,Y 587.786,Z 367.83,A -85,B 0,C 180,E1 -1542.296,E2 -1542.296} C_VEL
LIN {X 0,Y 587.682,Z 273.252,A -85,B 0,C 180,E1 -1543.459,E2 -1543.459} C_VEL
LIN {X 0,Y 587.384,Z 271.3,A -85,B 0,C 180,E1 -1543.513,E2 -1543.513} C_VEL
LIN {X 0,Y 587.476,Z 255.545,A -85,B 0,C 180,E1 -1545.792,E2 -1545.792} C_VEL
LIN {X 0,Y 587.588,Z 237.446,A -85,B 0,C 180,E1 -1548.478,E2 -1548.478} C_VEL
LIN {X 0,Y 587.723,Z 219.807,A -85,B 0,C 180,E1 -1551.135,E2 -1551.135} C_VEL
LIN {X 0,Y 587.46,Z 214.533,A -85,B 0,C 180,E1 -1551.952,E2 -1551.952} C_VEL
LIN {X 0,Y 587.321,Z 213.877,A -85,B 0,C 180,E1 -1552.143,E2 -1552.143} C_VEL
LIN {X 0,Y 587.315,Z 213.821,A -85,B 0,C 180,E1 -1554.759,E2 -1554.759} C_VEL
LIN {X 0,Y 587.33,Z 213.82,A -85,B 0,C 180,E1 -1557.045,E2 -1557.045} C_VEL
LIN {X 0,Y 587.338,Z 213.821,A -85,B 0,C 180,E1 -1559.378,E2 -1559.378} C_VEL
LIN {X 0,Y 587.349,Z 213.826,A -85,B 0,C 180,E1 -1561.835,E2 -1561.835} C_VEL
LIN {X 0,Y 587.34,Z 213.821,A -85,B 0,C 180,E1 -1564.345,E2 -1564.345} C_VEL
LIN {X 0,Y 587.341,Z 213.82,A -85,B 0,C 180,E1 -1567.606,E2 -1567.606} C_VEL
LIN {X 0,Y 587.306,Z 213.83,A -85,B 0,C 180,E1 -1570.253,E2 -1570.253} C_VEL
LIN {X 0,Y 587.299,Z 213.822,A -85,B 0,C 180,E1 -1573.115,E2 -1573.115} C_VEL
LIN {X 0,Y 587.309,Z 213.827,A -85,B 0,C 180,E1 -1576.047,E2 -1576.047} C_VEL
LIN {X 0,Y 587.327,Z 213.821,A -85,B 0,C 180,E1 -1578.924,E2 -1578.924} C_VEL
LIN {X 0,Y 587.312,Z 213.82,A -85,B 0,C 180,E1 -1581.518,E2 -1581.518} C_VEL
LIN {X 0,Y 587.282,Z 213.827,A -85,B 0,C 180,E1 -1584.098,E2 -1584.098} C_VEL
LIN {X 0,Y 587.327,Z 213.829,A -85,B 0,C 180,E1 -1586.601,E2 -1586.601} C_VEL
LIN {X 0,Y 587.313,Z 213.825,A -85,B 0,C 180,E1 -1589.031,E2 -1589.031} C_VEL
LIN {X 0,Y 587.299,Z 213.823,A -85,B 0,C 180,E1 -1591.4,E2 -1591.4} C_VEL
LIN {X 0,Y 587.298,Z 213.822,A -85,B 0,C 180,E1 -1593.828,E2 -1593.828} C_VEL
LIN {X 0,Y 587.293,Z 213.831,A -85,B 0,C 180,E1 -1596.738,E2 -1596.738} C_VEL
LIN {X 0,Y 587.299,Z 213.822,A -85,B 0,C 180,E1 -1599.692,E2 -1599.692} C_VEL
LIN {X 0,Y 587.273,Z 213.825,A -85,B 0,C 180,E1 -1601.87,E2 -1601.87} C_VEL
LIN {X 0,Y 587.287,Z 213.823,A -85,B 0,C 180,E1 -1604.022,E2 -1604.022} C_VEL
LIN {X 0,Y 587.287,Z 213.829,A -85,B 0,C 180,E1 -1606.855,E2 -1606.855} C_VEL
LIN {X 0,Y 587.285,Z 213.827,A -85,B 0,C 180,E1 -1609.657,E2 -1609.657} C_VEL
LIN {X 0,Y 587.289,Z 213.822,A -85,B 0,C 180,E1 -1612.434,E2 -1612.434} C_VEL
LIN {X 0,Y 587.351,Z 213.823,A -85,B 0,C 180,E1 -1615.193,E2 -1615.193} C_VEL
LIN {X 0,Y 587.32,Z 213.822,A -85,B 0,C 180,E1 -1617.94,E2 -1617.94} C_VEL
LIN {X 0,Y 587.338,Z 213.82,A -85,B 0,C 180,E1 -1619.997,E2 -1619.997} C_VEL
LIN {X 0,Y 587.315,Z 213.82,A -85,B 0,C 180,E1 -1622.741,E2 -1622.741} C_VEL
LIN {X 0,Y 587.32,Z 213.827,A -85,B 0,C 180,E1 -1625.49,E2 -1625.49} C_VEL
LIN {X 0,Y 587.314,Z 213.822,A -85,B 0,C 180,E1 -1628.253,E2 -1628.253} C_VEL
LIN {X 0,Y 587.309,Z 213.821,A -85,B 0,C 180,E1 -1631.122,E2 -1631.122} C_VEL
LIN {X 0,Y 587.32,Z 213.825,A -85,B 0,C 180,E1 -1634.249,E2 -1634.249} C_VEL
LIN {X 0,Y 587.301,Z 213.821,A -85,B 0,C 180,E1 -1636.804,E2 -1636.804} C_VEL
LIN {X 0,Y 587.275,Z 213.832,A -85,B 0,C 180,E1 -1638.262,E2 -1638.262} C_VEL
LIN {X 0,Y 586.629,Z 213.908,A -85,B 0,C 180,E1 -1638.834,E2 -1638.834} C_VEL
LIN {X 0,Y 583.816,Z 214.261,A -85,B 0,C 180,E1 -1639.763,E2 -1639.763} C_VEL
LIN {X 0,Y 581.415,Z 214.559,A -85,B 0,C 180,E1 -1640.51,E2 -1640.51} C_VEL
LIN {X 0,Y 580.36,Z 214.687,A -85,B 0,C 180,E1 -1641.087,E2 -1641.087} C_VEL
LIN {X 0,Y 580.261,Z 214.699,A -85,B 0,C 180,E1 -1641.282,E2 -1641.282} C_VEL
LIN {X 0,Y 580.247,Z 214.702,A -85,B 0,C 180,E1 -1643.555,E2 -1643.555} C_VEL
LIN {X 0,Y 580.248,Z 214.704,A -85,B 0,C 180,E1 -1645.847,E2 -1645.847} C_VEL
LIN {X 0,Y 580.269,Z 214.706,A -85,B 0,C 180,E1 -1648.183,E2 -1648.183} C_VEL
LIN {X 0,Y 580.253,Z 214.705,A -85,B 0,C 180,E1 -1650.692,E2 -1650.692} C_VEL
LIN {X 0,Y 580.269,Z 214.698,A -85,B 0,C 180,E1 -1653.314,E2 -1653.314} C_VEL
LIN {X 0,Y 580.295,Z 214.694,A -85,B 0,C 180,E1 -1655.766,E2 -1655.766} C_VEL
LIN {X 0,Y 580.256,Z 214.703,A -85,B 0,C 180,E1 -1658.144,E2 -1658.144} C_VEL
LIN {X 0,Y 580.287,Z 214.704,A -85,B 0,C 180,E1 -1660.839,E2 -1660.839} C_VEL
LIN {X 0,Y 580.254,Z 214.7,A -85,B 0,C 180,E1 -1663.654,E2 -1663.654} C_VEL
LIN {X 0,Y 580.256,Z 214.708,A -85,B 0,C 180,E1 -1666.605,E2 -1666.605} C_VEL
LIN {X 0,Y 580.303,Z 214.831,A -85,B 0,C 180,E1 -1668.438,E2 -1668.438} C_VEL
LIN {X 0,Y 580.63,Z 219.082,A -85,B 0,C 180,E1 -1669.187,E2 -1669.187} C_VEL
LIN {X 0,Y 580.45,Z 236.734,A -85,B 0,C 180,E1 -1672.111,E2 -1672.111} C_VEL
LIN {X 0,Y 580.327,Z 255.027,A -85,B 0,C 180,E1 -1675.097,E2 -1675.097} C_VEL
LIN {X 0,Y 580.395,Z 257.176,A -85,B 0,C 180,E1 -1675.385,E2 -1675.385} C_VEL
LIN {X 0,Y 580.935,Z 262.636,A -85,B 0,C 180,E1 -1675.481,E2 -1675.481} C_VEL
LIN {X 0,Y 580.792,Z 364.727,A -85,B 0,C 180,E1 -1676.768,E2 -1676.768} C_VEL
LIN {X 0,Y 580.754,Z 378.399,A -85,B 0,C 180,E1 -1677.097,E2 -1677.097} C_VEL
LIN {X 0,Y 580.645,Z 390.229,A -85,B 0,C 180,E1 -1677.515,E2 -1677.515} C_VEL
LIN {X 0,Y 580.556,Z 401.044,A -85,B 0,C 180,E1 -1678.022,E2 -1678.022} C_VEL
LIN {X 0,Y 580.441,Z 412.609,A -85,B 0,C 180,E1 -1678.717,E2 -1678.717} C_VEL
LIN {X 0,Y 580.349,Z 423.389,A -85,B 0,C 180,E1 -1679.53,E2 -1679.53} C_VEL
LIN {X 0,Y 580.28,Z 432.28,A -85,B 0,C 180,E1 -1680.36,E2 -1680.36} C_VEL
LIN {X 0,Y 580.208,Z 440.01,A -85,B 0,C 180,E1 -1681.219,E2 -1681.219} C_VEL
LIN {X 0,Y 580.175,Z 446.928,A -85,B 0,C 180,E1 -1682.154,E2 -1682.154} C_VEL
LIN {X 0,Y 580.115,Z 454.093,A -85,B 0,C 180,E1 -1683.37,E2 -1683.37} C_VEL
LIN {X 0,Y 580.081,Z 459.368,A -85,B 0,C 180,E1 -1684.527,E2 -1684.527} C_VEL
LIN {X 0,Y 580.04,Z 463.268,A -85,B 0,C 180,E1 -1685.674,E2 -1685.674} C_VEL
LIN {X 0,Y 580.047,Z 466.32,A -85,B 0,C 180,E1 -1687.036,E2 -1687.036} C_VEL
LIN {X 0,Y 580.027,Z 467.498,A -85,B 0,C 180,E1 -1687.939,E2 -1687.939} C_VEL
LIN {X 0,Y 580.035,Z 467.971,A -85,B 0,C 180,E1 -1688.889,E2 -1688.889} C_VEL
LIN {X 0,Y 580.045,Z 467.479,A -85,B 0,C 180,E1 -1690.17,E2 -1690.17} C_VEL
LIN {X 0,Y 580.047,Z 466.554,A -85,B 0,C 180,E1 -1690.906,E2 -1690.906} C_VEL
LIN {X 0,Y 580.037,Z 465.202,A -85,B 0,C 180,E1 -1691.639,E2 -1691.639} C_VEL
LIN {X 0,Y 580.072,Z 462.3,A -85,B 0,C 180,E1 -1692.734,E2 -1692.734} C_VEL
LIN {X 0,Y 580.106,Z 458.309,A -85,B 0,C 180,E1 -1693.822,E2 -1693.822} C_VEL
LIN {X 0,Y 580.116,Z 453.14,A -85,B 0,C 180,E1 -1694.903,E2 -1694.903} C_VEL
LIN {X 0,Y 580.173,Z 446.623,A -85,B 0,C 180,E1 -1695.981,E2 -1695.981} C_VEL
LIN {X 0,Y 580.217,Z 438.478,A -85,B 0,C 180,E1 -1697.052,E2 -1697.052} C_VEL
LIN {X 0,Y 580.298,Z 428.36,A -85,B 0,C 180,E1 -1698.12,E2 -1698.12} C_VEL
LIN {X 0,Y 580.399,Z 417.759,A -85,B 0,C 180,E1 -1699.007,E2 -1699.007} C_VEL
LIN {X 0,Y 580.486,Z 407.279,A -85,B 0,C 180,E1 -1699.714,E2 -1699.714} C_VEL
LIN {X 0,Y 580.62,Z 395.732,A -85,B 0,C 180,E1 -1700.333,E2 -1700.333} C_VEL
LIN {X 0,Y 580.714,Z 383.814,A -85,B 0,C 180,E1 -1700.818,E2 -1700.818} C_VEL
LIN {X 0,Y 580.756,Z 371.01,A -85,B 0,C 180,E1 -1701.191,E2 -1701.191} C_VEL
LIN {X 0,Y 580.841,Z 357.397,A -85,B 0,C 180,E1 -1701.434,E2 -1701.434} C_VEL
LIN {X 0,Y 580.875,Z 260.807,A -85,B 0,C 180,E1 -1702.633,E2 -1702.633} C_VEL
LIN {X 0,Y 580.333,Z 256.927,A -85,B 0,C 180,E1 -1702.721,E2 -1702.721} C_VEL
LIN {X 0,Y 580.419,Z 239.735,A -85,B 0,C 180,E1 -1705.487,E2 -1705.487} C_VEL
LIN {X 0,Y 580.542,Z 224.992,A -85,B 0,C 180,E1 -1707.92,E2 -1707.92} C_VEL
LIN {X 0,Y 580.607,Z 216.675,A -85,B 0,C 180,E1 -1709.308,E2 -1709.308} C_VEL
LIN {X 0,Y 580.311,Z 214.824,A -85,B 0,C 180,E1 -1709.654,E2 -1709.654} C_VEL
LIN {X 0,Y 580.282,Z 214.698,A -85,B 0,C 180,E1 -1712.083,E2 -1712.083} C_VEL
LIN {X 0,Y 580.294,Z 214.698,A -85,B 0,C 180,E1 -1714.864,E2 -1714.864} C_VEL
LIN {X 0,Y 580.298,Z 214.701,A -85,B 0,C 180,E1 -1717.657,E2 -1717.657} C_VEL
LIN {X 0,Y 580.251,Z 214.7,A -85,B 0,C 180,E1 -1720.469,E2 -1720.469} C_VEL
LIN {X 0,Y 580.259,Z 214.699,A -85,B 0,C 180,E1 -1722.593,E2 -1722.593} C_VEL
LIN {X 0,Y 580.238,Z 214.701,A -85,B 0,C 180,E1 -1724.737,E2 -1724.737} C_VEL
LIN {X 0,Y 580.258,Z 214.707,A -85,B 0,C 180,E1 -1727.627,E2 -1727.627} C_VEL
LIN {X 0,Y 580.26,Z 214.709,A -85,B 0,C 180,E1 -1729.825,E2 -1729.825} C_VEL
LIN {X 0,Y 580.249,Z 214.7,A -85,B 0,C 180,E1 -1732.805,E2 -1732.805} C_VEL
LIN {X 0,Y 580.262,Z 214.698,A -85,B 0,C 180,E1 -1735.083,E2 -1735.083} C_VEL
LIN {X 0,Y 580.241,Z 214.711,A -85,B 0,C 180,E1 -1738.19,E2 -1738.19} C_VEL
LIN {X 0,Y 580.251,Z 214.703,A -85,B 0,C 180,E1 -1740.698,E2 -1740.698} C_VEL
LIN {X 0,Y 580.245,Z 214.7,A -85,B 0,C 180,E1 -1743.316,E2 -1743.316} C_VEL
LIN {X 0,Y 580.194,Z 214.708,A -85,B 0,C 180,E1 -1745.757,E2 -1745.757} C_VEL
LIN {X 0,Y 580.245,Z 214.706,A -85,B 0,C 180,E1 -1748.151,E2 -1748.151} C_VEL
LIN {X 0,Y 580.249,Z 214.706,A -85,B 0,C 180,E1 -1750.849,E2 -1750.849} C_VEL
LIN {X 0,Y 580.214,Z 214.705,A -85,B 0,C 180,E1 -1753.39,E2 -1753.39} C_VEL
LIN {X 0,Y 580.244,Z 214.705,A -85,B 0,C 180,E1 -1756.345,E2 -1756.345} C_VEL
LIN {X 0,Y 580.273,Z 214.702,A -85,B 0,C 180,E1 -1759.16,E2 -1759.16} C_VEL
LIN {X 0,Y 580.261,Z 214.698,A -85,B 0,C 180,E1 -1761.932,E2 -1761.932} C_VEL
LIN {X 0,Y 580.229,Z 214.705,A -85,B 0,C 180,E1 -1764.456,E2 -1764.456} C_VEL
LIN {X 0,Y 580.266,Z 214.707,A -85,B 0,C 180,E1 -1766.978,E2 -1766.978} C_VEL
LIN {X 0,Y 580.256,Z 214.705,A -85,B 0,C 180,E1 -1769.427,E2 -1769.427} C_VEL
LIN {X 0,Y 580.236,Z 214.701,A -85,B 0,C 180,E1 -1772.154,E2 -1772.154} C_VEL
LIN {X 0,Y 580.23,Z 214.706,A -85,B 0,C 180,E1 -1774.921,E2 -1774.921} C_VEL
LIN {X 0,Y 580.276,Z 214.704,A -85,B 0,C 180,E1 -1777.201,E2 -1777.201} C_VEL
LIN {X 0,Y 580.262,Z 214.709,A -85,B 0,C 180,E1 -1779.44,E2 -1779.44} C_VEL
LIN {X 0,Y 580.243,Z 214.71,A -85,B 0,C 180,E1 -1781.648,E2 -1781.648} C_VEL
LIN {X 0,Y 580.266,Z 214.698,A -85,B 0,C 180,E1 -1784.55,E2 -1784.55} C_VEL
LIN {X 0,Y 580.247,Z 214.7,A -85,B 0,C 180,E1 -1786.699,E2 -1786.699} C_VEL
LIN {X 0,Y 580.267,Z 214.697,A -85,B 0,C 180,E1 -1788.829,E2 -1788.829} C_VEL
LIN {X 0,Y 580.302,Z 214.7,A -85,B 0,C 180,E1 -1791.647,E2 -1791.647} C_VEL
LIN {X 0,Y 580.304,Z 214.696,A -85,B 0,C 180,E1 -1794.443,E2 -1794.443} C_VEL
LIN {X 0,Y 580.335,Z 214.697,A -85,B 0,C 180,E1 -1797.921,E2 -1797.921} C_VEL
LIN {X 0,Y 580.357,Z 214.689,A -85,B 0,C 180,E1 -1800.697,E2 -1800.697} C_VEL
LIN {X 0,Y 580.332,Z 214.692,A -85,B 0,C 180,E1 -1802.779,E2 -1802.779} C_VEL
LIN {X 0,Y 580.295,Z 214.695,A -85,B 0,C 180,E1 -1805.563,E2 -1805.563} C_VEL
LIN {X 0,Y 580.297,Z 214.704,A -85,B 0,C 180,E1 -1808.359,E2 -1808.359} C_VEL
LIN {X 0,Y 580.312,Z 214.693,A -85,B 0,C 180,E1 -1811.193,E2 -1811.193} C_VEL
LIN {X 0,Y 580.302,Z 214.695,A -85,B 0,C 180,E1 -1814.02,E2 -1814.02} C_VEL
LIN {X 0,Y 580.302,Z 214.701,A -85,B 0,C 180,E1 -1816.908,E2 -1816.908} C_VEL
LIN {X 0,Y 580.284,Z 214.695,A -85,B 0,C 180,E1 -1819.825,E2 -1819.825} C_VEL
LIN {X 0,Y 580.26,Z 214.699,A -85,B 0,C 180,E1 -1822.055,E2 -1822.055} C_VEL
LIN {X 0,Y 580.289,Z 214.704,A -85,B 0,C 180,E1 -1825.082,E2 -1825.082} C_VEL
LIN {X 0,Y 580.254,Z 214.7,A -85,B 0,C 180,E1 -1827.849,E2 -1827.849} C_VEL
LIN {X 0,Y 580.279,Z 214.699,A -85,B 0,C 180,E1 -1830.692,E2 -1830.692} C_VEL
LIN {X 0,Y 580.291,Z 214.705,A -85,B 0,C 180,E1 -1833.313,E2 -1833.313} C_VEL
LIN {X 0,Y 580.239,Z 214.705,A -85,B 0,C 180,E1 -1835.754,E2 -1835.754} C_VEL
LIN {X 0,Y 580.293,Z 214.695,A -85,B 0,C 180,E1 -1838.148,E2 -1838.148} C_VEL
LIN {X 0,Y 580.291,Z 214.696,A -85,B 0,C 180,E1 -1840.846,E2 -1840.846} C_VEL
LIN {X 0,Y 580.248,Z 214.71,A -85,B 0,C 180,E1 -1843.662,E2 -1843.662} C_VEL
LIN {X 0,Y 580.246,Z 214.7,A -85,B 0,C 180,E1 -1846.614,E2 -1846.614} C_VEL
LIN {X 0,Y 580.289,Z 214.697,A -85,B 0,C 180,E1 -1849.155,E2 -1849.155} C_VEL
LIN {X 0,Y 580.297,Z 214.704,A -85,B 0,C 180,E1 -1851.928,E2 -1851.928} C_VEL
LIN {X 0,Y 580.24,Z 214.704,A -85,B 0,C 180,E1 -1854.451,E2 -1854.451} C_VEL
LIN {X 0,Y 580.295,Z 214.694,A -85,B 0,C 180,E1 -1856.975,E2 -1856.975} C_VEL
LIN {X 0,Y 580.291,Z 214.696,A -85,B 0,C 180,E1 -1859.424,E2 -1859.424} C_VEL
LIN {X 0,Y 580.297,Z 214.705,A -85,B 0,C 180,E1 -1862.143,E2 -1862.143} C_VEL
LIN {X 0,Y 580.297,Z 214.697,A -85,B 0,C 180,E1 -1864.919,E2 -1864.919} C_VEL
LIN {X 0,Y 580.313,Z 214.892,A -85,B 0,C 180,E1 -1867.808,E2 -1867.808} C_VEL
LIN {X 0,Y 580.806,Z 219.451,A -85,B 0,C 180,E1 -1868.546,E2 -1868.546} C_VEL
LIN {X 0,Y 580.628,Z 238.637,A -85,B 0,C 180,E1 -1871.473,E2 -1871.473} C_VEL
LIN {X 0,Y 580.475,Z 256.736,A -85,B 0,C 180,E1 -1874.191,E2 -1874.191} C_VEL
LIN {X 0,Y 580.386,Z 271.265,A -85,B 0,C 180,E1 -1876.319,E2 -1876.319} C_VEL
LIN {X 0,Y 580.98,Z 276.429,A -85,B 0,C 180,E1 -1876.422,E2 -1876.422} C_VEL
LIN {X 0,Y 580.825,Z 378.895,A -85,B 0,C 180,E1 -1877.708,E2 -1877.708} C_VEL
LIN {X 0,Y 580.745,Z 392.185,A -85,B 0,C 180,E1 -1878.016,E2 -1878.016} C_VEL
LIN {X 0,Y 580.634,Z 404.349,A -85,B 0,C 180,E1 -1878.435,E2 -1878.435} C_VEL
LIN {X 0,Y 580.563,Z 416.61,A -85,B 0,C 180,E1 -1879.008,E2 -1879.008} C_VEL
LIN {X 0,Y 580.418,Z 428.187,A -85,B 0,C 180,E1 -1879.711,E2 -1879.711} C_VEL
LIN {X 0,Y 580.343,Z 438.588,A -85,B 0,C 180,E1 -1880.502,E2 -1880.502} C_VEL
LIN {X 0,Y 580.264,Z 447.051,A -85,B 0,C 180,E1 -1881.291,E2 -1881.291} C_VEL
LIN {X 0,Y 580.223,Z 454.952,A -85,B 0,C 180,E1 -1882.167,E2 -1882.167} C_VEL
LIN {X 0,Y 580.158,Z 462.635,A -85,B 0,C 180,E1 -1883.219,E2 -1883.219} C_VEL
LIN {X 0,Y 580.139,Z 469.675,A -85,B 0,C 180,E1 -1884.437,E2 -1884.437} C_VEL
LIN {X 0,Y 580.108,Z 474.368,A -85,B 0,C 180,E1 -1885.482,E2 -1885.482} C_VEL
LIN {X 0,Y 580.123,Z 477.954,A -85,B 0,C 180,E1 -1886.526,E2 -1886.526} C_VEL
LIN {X 0,Y 580.043,Z 479.806,A -85,B 0,C 180,E1 -1887.221,E2 -1887.221} C_VEL
LIN {X 0,Y 580.038,Z 481.197,A -85,B 0,C 180,E1 -1887.916,E2 -1887.916} C_VEL
LIN {X 0,Y 580.04,Z 482.784,A -85,B 0,C 180,E1 -1889.305,E2 -1889.305} C_VEL
LIN {X 0,Y 580.037,Z 483,A -85,B 0,C 180,E1 -1889.999,E2 -1889.999} C_VEL
LIN {X 0,Y 580.046,Z 482.187,A -85,B 0,C 180,E1 -1891.387,E2 -1891.387} C_VEL
LIN {X 0,Y 580.038,Z 481.202,A -85,B 0,C 180,E1 -1892.082,E2 -1892.082} C_VEL
LIN {X 0,Y 580.043,Z 479.812,A -85,B 0,C 180,E1 -1892.777,E2 -1892.777} C_VEL
LIN {X 0,Y 580.109,Z 476.899,A -85,B 0,C 180,E1 -1893.819,E2 -1893.819} C_VEL
LIN {X 0,Y 580.053,Z 472.954,A -85,B 0,C 180,E1 -1894.864,E2 -1894.864} C_VEL
LIN {X 0,Y 580.14,Z 466.883,A -85,B 0,C 180,E1 -1896.084,E2 -1896.084} C_VEL
LIN {X 0,Y 580.184,Z 460.246,A -85,B 0,C 180,E1 -1897.131,E2 -1897.131} C_VEL
LIN {X 0,Y 580.246,Z 452,A -85,B 0,C 180,E1 -1898.181,E2 -1898.181} C_VEL
LIN {X 0,Y 580.332,Z 441.615,A -85,B 0,C 180,E1 -1899.232,E2 -1899.232} C_VEL
LIN {X 0,Y 580.434,Z 430.763,A -85,B 0,C 180,E1 -1900.111,E2 -1900.111} C_VEL
LIN {X 0,Y 580.537,Z 419.804,A -85,B 0,C 180,E1 -1900.814,E2 -1900.814} C_VEL
LIN {X 0,Y 580.663,Z 407.57,A -85,B 0,C 180,E1 -1901.428,E2 -1901.428} C_VEL
LIN {X 0,Y 580.731,Z 395.906,A -85,B 0,C 180,E1 -1901.871,E2 -1901.871} C_VEL
LIN {X 0,Y 580.787,Z 383.567,A -85,B 0,C 180,E1 -1902.202,E2 -1902.202} C_VEL
LIN {X 0,Y 580.87,Z 367.83,A -85,B 0,C 180,E1 -1902.445,E2 -1902.445} C_VEL
LIN {X 0,Y 580.903,Z 274.819,A -85,B 0,C 180,E1 -1903.6,E2 -1903.6} C_VEL
LIN {X 0,Y 580.386,Z 271.311,A -85,B 0,C 180,E1 -1903.679,E2 -1903.679} C_VEL
LIN {X 0,Y 580.487,Z 255.545,A -85,B 0,C 180,E1 -1905.987,E2 -1905.987} C_VEL
LIN {X 0,Y 580.614,Z 237.446,A -85,B 0,C 180,E1 -1908.708,E2 -1908.708} C_VEL
LIN {X 0,Y 580.835,Z 219.466,A -85,B 0,C 180,E1 -1911.45,E2 -1911.45} C_VEL
LIN {X 0,Y 580.316,Z 214.888,A -85,B 0,C 180,E1 -1912.19,E2 -1912.19} C_VEL
LIN {X 0,Y 580.291,Z 214.698,A -85,B 0,C 180,E1 -1915.079,E2 -1915.079} C_VEL
LIN {X 0,Y 580.297,Z 214.705,A -85,B 0,C 180,E1 -1917.857,E2 -1917.857} C_VEL
LIN {X 0,Y 580.28,Z 214.697,A -85,B 0,C 180,E1 -1920.692,E2 -1920.692} C_VEL
LIN {X 0,Y 580.302,Z 214.695,A -85,B 0,C 180,E1 -1923.315,E2 -1923.315} C_VEL
LIN {X 0,Y 580.242,Z 214.707,A -85,B 0,C 180,E1 -1925.754,E2 -1925.754} C_VEL
LIN {X 0,Y 580.283,Z 214.705,A -85,B 0,C 180,E1 -1928.145,E2 -1928.145} C_VEL
LIN {X 0,Y 580.292,Z 214.696,A -85,B 0,C 180,E1 -1930.842,E2 -1930.842} C_VEL
LIN {X 0,Y 580.267,Z 214.7,A -85,B 0,C 180,E1 -1933.657,E2 -1933.657} C_VEL
LIN {X 0,Y 580.262,Z 214.703,A -85,B 0,C 180,E1 -1936.609,E2 -1936.609} C_VEL
LIN {X 0,Y 580.29,Z 214.696,A -85,B 0,C 180,E1 -1939.154,E2 -1939.154} C_VEL
LIN {X 0,Y 580.281,Z 214.698,A -85,B 0,C 180,E1 -1941.926,E2 -1941.926} C_VEL
LIN {X 0,Y 580.243,Z 214.71,A -85,B 0,C 180,E1 -1944.45,E2 -1944.45} C_VEL
LIN {X 0,Y 580.281,Z 214.7,A -85,B 0,C 180,E1 -1946.973,E2 -1946.973} C_VEL
LIN {X 0,Y 580.274,Z 214.698,A -85,B 0,C 180,E1 -1949.422,E2 -1949.422} C_VEL
LIN {X 0,Y 580.254,Z 214.701,A -85,B 0,C 180,E1 -1952.146,E2 -1952.146} C_VEL
LIN {X 0,Y 580.275,Z 214.706,A -85,B 0,C 180,E1 -1954.917,E2 -1954.917} C_VEL
LIN {X 0,Y 580.244,Z 214.7,A -85,B 0,C 180,E1 -1957.944,E2 -1957.944} C_VEL
LIN {X 0,Y 580.289,Z 214.703,A -85,B 0,C 180,E1 -1960.847,E2 -1960.847} C_VEL
LIN {X 0,Y 580.24,Z 214.701,A -85,B 0,C 180,E1 -1963.822,E2 -1963.822} C_VEL
LIN {X 0,Y 580.24,Z 214.704,A -85,B 0,C 180,E1 -1966.693,E2 -1966.693} C_VEL
LIN {X 0,Y 580.295,Z 214.698,A -85,B 0,C 180,E1 -1968.824,E2 -1968.824} C_VEL
LIN {X 0,Y 580.274,Z 214.701,A -85,B 0,C 180,E1 -1971.641,E2 -1971.641} C_VEL
LIN {X 0,Y 580.24,Z 214.705,A -85,B 0,C 180,E1 -1973.739,E2 -1973.739} C_VEL
LIN {X 0,Y 580.223,Z 214.706,A -85,B 0,C 180,E1 -1975.83,E2 -1975.83} C_VEL
LIN {X 0,Y 580.295,Z 214.698,A -85,B 0,C 180,E1 -1977.915,E2 -1977.915} C_VEL
LIN {X 0,Y 580.31,Z 214.695,A -85,B 0,C 180,E1 -1979.997,E2 -1979.997} C_VEL
LIN {X 0,Y 580.286,Z 214.696,A -85,B 0,C 180,E1 -1982.774,E2 -1982.774} C_VEL
LIN {X 0,Y 580.286,Z 214.704,A -85,B 0,C 180,E1 -1985.557,E2 -1985.557} C_VEL
LIN {X 0,Y 580.282,Z 214.697,A -85,B 0,C 180,E1 -1988.354,E2 -1988.354} C_VEL
LIN {X 0,Y 580.28,Z 214.698,A -85,B 0,C 180,E1 -1991.188,E2 -1991.188} C_VEL
LIN {X 0,Y 580.276,Z 214.701,A -85,B 0,C 180,E1 -1994.329,E2 -1994.329} C_VEL
LIN {X 0,Y 580.265,Z 214.698,A -85,B 0,C 180,E1 -1996.903,E2 -1996.903} C_VEL
LIN {X 0,Y 580.26,Z 214.705,A -85,B 0,C 180,E1 -1999.82,E2 -1999.82} C_VEL
LIN {X 0,Y 580.261,Z 214.699,A -85,B 0,C 180,E1 -2001.282,E2 -2001.282} C_VEL
LIN {X 0,Y 579.555,Z 214.795,A -85,B 0,C 180,E1 -2001.861,E2 -2001.861} C_VEL
LIN {X 0,Y 576.675,Z 215.149,A -85,B 0,C 180,E1 -2002.801,E2 -2002.801} C_VEL
LIN {X 0,Y 574.283,Z 215.446,A -85,B 0,C 180,E1 -2003.557,E2 -2003.557} C_VEL
LIN {X 0,Y 573.283,Z 215.578,A -85,B 0,C 180,E1 -2004.141,E2 -2004.141} C_VEL
LIN {X 0,Y 573.216,Z 215.579,A -85,B 0,C 180,E1 -2004.339,E2 -2004.339} C_VEL
LIN {X 0,Y 573.186,Z 215.581,A -85,B 0,C 180,E1 -2006.975,E2 -2006.975} C_VEL
LIN {X 0,Y 573.218,Z 215.575,A -85,B 0,C 180,E1 -2009.486,E2 -2009.486} C_VEL
LIN {X 0,Y 573.225,Z 215.582,A -85,B 0,C 180,E1 -2012.642,E2 -2012.642} C_VEL
LIN {X 0,Y 573.238,Z 215.574,A -85,B 0,C 180,E1 -2015.181,E2 -2015.181} C_VEL
LIN {X 0,Y 573.203,Z 215.579,A -85,B 0,C 180,E1 -2017.805,E2 -2017.805} C_VEL
LIN {X 0,Y 573.232,Z 215.584,A -85,B 0,C 180,E1 -2020.526,E2 -2020.526} C_VEL
LIN {X 0,Y 573.218,Z 215.577,A -85,B 0,C 180,E1 -2023.668,E2 -2023.668} C_VEL
LIN {X 0,Y 573.217,Z 215.585,A -85,B 0,C 180,E1 -2026.641,E2 -2026.641} C_VEL
LIN {X 0,Y 573.273,Z 215.739,A -85,B 0,C 180,E1 -2028.375,E2 -2028.375} C_VEL
LIN {X 0,Y 573.65,Z 220.966,A -85,B 0,C 180,E1 -2029.266,E2 -2029.266} C_VEL
LIN {X 0,Y 573.442,Z 236.941,A -85,B 0,C 180,E1 -2031.932,E2 -2031.932} C_VEL
LIN {X 0,Y 573.28,Z 254.402,A -85,B 0,C 180,E1 -2034.819,E2 -2034.819} C_VEL
LIN {X 0,Y 573.33,Z 257.075,A -85,B 0,C 180,E1 -2035.207,E2 -2035.207} C_VEL
LIN {X 0,Y 574.038,Z 262.91,A -85,B 0,C 180,E1 -2035.318,E2 -2035.318} C_VEL
LIN {X 0,Y 573.878,Z 364.444,A -85,B 0,C 180,E1 -2036.612,E2 -2036.612} C_VEL
LIN {X 0,Y 573.79,Z 377.871,A -85,B 0,C 180,E1 -2036.934,E2 -2036.934} C_VEL
LIN {X 0,Y 573.697,Z 390.519,A -85,B 0,C 180,E1 -2037.385,E2 -2037.385} C_VEL
LIN {X 0,Y 573.559,Z 402.394,A -85,B 0,C 180,E1 -2037.961,E2 -2037.961} C_VEL
LIN {X 0,Y 573.409,Z 414.38,A -85,B 0,C 180,E1 -2038.712,E2 -2038.712} C_VEL
LIN {X 0,Y 573.332,Z 424.711,A -85,B 0,C 180,E1 -2039.525,E2 -2039.525} C_VEL
LIN {X 0,Y 573.21,Z 434.722,A -85,B 0,C 180,E1 -2040.509,E2 -2040.509} C_VEL
LIN {X 0,Y 573.131,Z 443.566,A -85,B 0,C 180,E1 -2041.586,E2 -2041.586} C_VEL
LIN {X 0,Y 573.062,Z 450.371,A -85,B 0,C 180,E1 -2042.621,E2 -2042.621} C_VEL
LIN {X 0,Y 573.017,Z 456.513,A -85,B 0,C 180,E1 -2043.8,E2 -2043.8} C_VEL
LIN {X 0,Y 572.999,Z 460.973,A -85,B 0,C 180,E1 -2044.909,E2 -2044.909} C_VEL
LIN {X 0,Y 572.944,Z 464.539,A -85,B 0,C 180,E1 -2046.123,E2 -2046.123} C_VEL
LIN {X 0,Y 572.939,Z 466.162,A -85,B 0,C 180,E1 -2046.913,E2 -2046.913} C_VEL
LIN {X 0,Y 572.934,Z 467.2,A -85,B 0,C 180,E1 -2047.651,E2 -2047.651} C_VEL
LIN {X 0,Y 572.947,Z 467.946,A -85,B 0,C 180,E1 -2048.774,E2 -2048.774} C_VEL
LIN {X 0,Y 572.962,Z 467.674,A -85,B 0,C 180,E1 -2049.914,E2 -2049.914} C_VEL
LIN {X 0,Y 572.943,Z 466.741,A -85,B 0,C 180,E1 -2050.81,E2 -2050.81} C_VEL
LIN {X 0,Y 572.954,Z 464.091,A -85,B 0,C 180,E1 -2052.143,E2 -2052.143} C_VEL
LIN {X 0,Y 573.009,Z 460.417,A -85,B 0,C 180,E1 -2053.339,E2 -2053.339} C_VEL
LIN {X 0,Y 573.021,Z 456.254,A -85,B 0,C 180,E1 -2054.347,E2 -2054.347} C_VEL
LIN {X 0,Y 573.068,Z 450.686,A -85,B 0,C 180,E1 -2055.414,E2 -2055.414} C_VEL
LIN {X 0,Y 573.097,Z 443.396,A -85,B 0,C 180,E1 -2056.527,E2 -2056.527} C_VEL
LIN {X 0,Y 573.216,Z 434.443,A -85,B 0,C 180,E1 -2057.611,E2 -2057.611} C_VEL
LIN {X 0,Y 573.334,Z 425.1,A -85,B 0,C 180,E1 -2058.529,E2 -2058.529} C_VEL
LIN {X 0,Y 573.438,Z 415.107,A -85,B 0,C 180,E1 -2059.327,E2 -2059.327} C_VEL
LIN {X 0,Y 573.533,Z 404.08,A -85,B 0,C 180,E1 -2060.034,E2 -2060.034} C_VEL
LIN {X 0,Y 573.67,Z 391.584,A -85,B 0,C 180,E1 -2060.659,E2 -2060.659} C_VEL
LIN {X 0,Y 573.759,Z 378.867,A -85,B 0,C 180,E1 -2061.127,E2 -2061.127} C_VEL
LIN {X 0,Y 573.896,Z 365.233,A -85,B 0,C 180,E1 -2061.462,E2 -2061.462} C_VEL
LIN {X 0,Y 573.937,Z 328.334,A -85,B 0,C 180,E1 -2061.95,E2 -2061.95} C_VEL
LIN {X 0,Y 573.82,Z 260.362,A -85,B 0,C 180,E1 -2062.809,E2 -2062.809} C_VEL
LIN {X 0,Y 573.34,Z 257.041,A -85,B 0,C 180,E1 -2062.884,E2 -2062.884} C_VEL
LIN {X 0,Y 573.333,Z 248.777,A -85,B 0,C 180,E1 -2064.197,E2 -2064.197} C_VEL
LIN {X 0,Y 573.543,Z 230.743,A -85,B 0,C 180,E1 -2067.192,E2 -2067.192} C_VEL
LIN {X 0,Y 573.658,Z 218.245,A -85,B 0,C 180,E1 -2069.299,E2 -2069.299} C_VEL
LIN {X 0,Y 573.273,Z 215.678,A -85,B 0,C 180,E1 -2069.782,E2 -2069.782} C_VEL
LIN {X 0,Y 573.254,Z 215.573,A -85,B 0,C 180,E1 -2072.109,E2 -2072.109} C_VEL
LIN {X 0,Y 573.267,Z 215.574,A -85,B 0,C 180,E1 -2074.924,E2 -2074.924} C_VEL
LIN {X 0,Y 573.246,Z 215.578,A -85,B 0,C 180,E1 -2077.752,E2 -2077.752} C_VEL
LIN {X 0,Y 573.218,Z 215.576,A -85,B 0,C 180,E1 -2080.599,E2 -2080.599} C_VEL
LIN {X 0,Y 573.219,Z 215.576,A -85,B 0,C 180,E1 -2082.751,E2 -2082.751} C_VEL
LIN {X 0,Y 573.186,Z 215.58,A -85,B 0,C 180,E1 -2084.922,E2 -2084.922} C_VEL
LIN {X 0,Y 573.209,Z 215.587,A -85,B 0,C 180,E1 -2087.851,E2 -2087.851} C_VEL
LIN {X 0,Y 573.208,Z 215.584,A -85,B 0,C 180,E1 -2090.079,E2 -2090.079} C_VEL
LIN {X 0,Y 573.195,Z 215.579,A -85,B 0,C 180,E1 -2093.102,E2 -2093.102} C_VEL
LIN {X 0,Y 573.201,Z 215.579,A -85,B 0,C 180,E1 -2095.414,E2 -2095.414} C_VEL
LIN {X 0,Y 573.187,Z 215.583,A -85,B 0,C 180,E1 -2098.568,E2 -2098.568} C_VEL
LIN {X 0,Y 573.191,Z 215.58,A -85,B 0,C 180,E1 -2100.996,E2 -2100.996} C_VEL
LIN {X 0,Y 573.207,Z 215.577,A -85,B 0,C 180,E1 -2103.524,E2 -2103.524} C_VEL
LIN {X 0,Y 573.154,Z 215.589,A -85,B 0,C 180,E1 -2106.057,E2 -2106.057} C_VEL
LIN {X 0,Y 573.199,Z 215.585,A -85,B 0,C 180,E1 -2108.706,E2 -2108.706} C_VEL
LIN {X 0,Y 573.175,Z 215.581,A -85,B 0,C 180,E1 -2111.463,E2 -2111.463} C_VEL
LIN {X 0,Y 573.181,Z 215.58,A -85,B 0,C 180,E1 -2113.669,E2 -2113.669} C_VEL
LIN {X 0,Y 573.205,Z 215.587,A -85,B 0,C 180,E1 -2116.644,E2 -2116.644} C_VEL
LIN {X 0,Y 573.223,Z 215.576,A -85,B 0,C 180,E1 -2119.479,E2 -2119.479} C_VEL
LIN {X 0,Y 573.208,Z 215.578,A -85,B 0,C 180,E1 -2122.196,E2 -2122.196} C_VEL
LIN {X 0,Y 573.215,Z 215.583,A -85,B 0,C 180,E1 -2125.233,E2 -2125.233} C_VEL
LIN {X 0,Y 573.209,Z 215.577,A -85,B 0,C 180,E1 -2128.187,E2 -2128.187} C_VEL
LIN {X 0,Y 573.222,Z 215.577,A -85,B 0,C 180,E1 -2130.636,E2 -2130.636} C_VEL
LIN {X 0,Y 573.186,Z 215.587,A -85,B 0,C 180,E1 -2133.519,E2 -2133.519} C_VEL
LIN {X 0,Y 573.198,Z 215.579,A -85,B 0,C 180,E1 -2136.137,E2 -2136.137} C_VEL
LIN {X 0,Y 573.241,Z 215.578,A -85,B 0,C 180,E1 -2139.177,E2 -2139.177} C_VEL
LIN {X 0,Y 573.2,Z 215.586,A -85,B 0,C 180,E1 -2141.414,E2 -2141.414} C_VEL
LIN {X 0,Y 573.206,Z 215.578,A -85,B 0,C 180,E1 -2144.355,E2 -2144.355} C_VEL
LIN {X 0,Y 573.208,Z 215.577,A -85,B 0,C 180,E1 -2146.532,E2 -2146.532} C_VEL
LIN {X 0,Y 573.239,Z 215.577,A -85,B 0,C 180,E1 -2149.406,E2 -2149.406} C_VEL
LIN {X 0,Y 573.222,Z 215.58,A -85,B 0,C 180,E1 -2152.252,E2 -2152.252} C_VEL
LIN {X 0,Y 573.277,Z 215.568,A -85,B 0,C 180,E1 -2155.08,E2 -2155.08} C_VEL
LIN {X 0,Y 573.306,Z 215.572,A -85,B 0,C 180,E1 -2157.895,E2 -2157.895} C_VEL
LIN {X 0,Y 573.328,Z 215.564,A -85,B 0,C 180,E1 -2160.705,E2 -2160.705} C_VEL
LIN {X 0,Y 573.296,Z 215.568,A -85,B 0,C 180,E1 -2162.813,E2 -2162.813} C_VEL
LIN {X 0,Y 573.264,Z 215.571,A -85,B 0,C 180,E1 -2165.631,E2 -2165.631} C_VEL
LIN {X 0,Y 573.243,Z 215.583,A -85,B 0,C 180,E1 -2168.463,E2 -2168.463} C_VEL
LIN {X 0,Y 573.283,Z 215.568,A -85,B 0,C 180,E1 -2171.314,E2 -2171.314} C_VEL
LIN {X 0,Y 573.266,Z 215.577,A -85,B 0,C 180,E1 -2174.415,E2 -2174.415} C_VEL
LIN {X 0,Y 573.257,Z 215.575,A -85,B 0,C 180,E1 -2177.114,E2 -2177.114} C_VEL
LIN {X 0,Y 573.241,Z 215.573,A -85,B 0,C 180,E1 -2180.079,E2 -2180.079} C_VEL
LIN {X 0,Y 573.229,Z 215.577,A -85,B 0,C 180,E1 -2182.34,E2 -2182.34} C_VEL
LIN {X 0,Y 573.238,Z 215.577,A -85,B 0,C 180,E1 -2185.413,E2 -2185.413} C_VEL
LIN {X 0,Y 573.211,Z 215.576,A -85,B 0,C 180,E1 -2188.02,E2 -2188.02} C_VEL
LIN {X 0,Y 573.239,Z 215.573,A -85,B 0,C 180,E1 -2190.178,E2 -2190.178} C_VEL
LIN {X 0,Y 573.257,Z 215.573,A -85,B 0,C 180,E1 -2192.647,E2 -2192.647} C_VEL
LIN {X 0,Y 573.201,Z 215.587,A -85,B 0,C 180,E1 -2195.19,E2 -2195.19} C_VEL
LIN {X 0,Y 573.239,Z 215.577,A -85,B 0,C 180,E1 -2197.809,E2 -2197.809} C_VEL
LIN {X 0,Y 573.258,Z 215.571,A -85,B 0,C 180,E1 -2200.526,E2 -2200.526} C_VEL
LIN {X 0,Y 573.211,Z 215.584,A -85,B 0,C 180,E1 -2203.363,E2 -2203.363} C_VEL
LIN {X 0,Y 573.217,Z 215.577,A -85,B 0,C 180,E1 -2206.336,E2 -2206.336} C_VEL
LIN {X 0,Y 573.217,Z 215.576,A -85,B 0,C 180,E1 -2208.541,E2 -2208.541} C_VEL
LIN {X 0,Y 573.245,Z 215.575,A -85,B 0,C 180,E1 -2211.298,E2 -2211.298} C_VEL
LIN {X 0,Y 573.198,Z 215.587,A -85,B 0,C 180,E1 -2214.022,E2 -2214.022} C_VEL
LIN {X 0,Y 573.262,Z 215.573,A -85,B 0,C 180,E1 -2216.516,E2 -2216.516} C_VEL
LIN {X 0,Y 573.23,Z 215.574,A -85,B 0,C 180,E1 -2219.119,E2 -2219.119} C_VEL
LIN {X 0,Y 573.251,Z 215.58,A -85,B 0,C 180,E1 -2221.973,E2 -2221.973} C_VEL
LIN {X 0,Y 573.244,Z 215.58,A -85,B 0,C 180,E1 -2224.588,E2 -2224.588} C_VEL
LIN {X 0,Y 573.28,Z 215.727,A -85,B 0,C 180,E1 -2227.663,E2 -2227.663} C_VEL
